LIN {X 0,Y 573.267,Z 626.574,A -85,B 0,C 180,E1 -2260.914,E2 -2260.914} C_VEL
LIN {X 0,Y 573.402,Z 606.241,A -85,B 0,C 180,E1 -2263.647,E2 -2263.647} C_VEL
LIN {X 0,Y 573.594,Z 585.071,A -85,B 0,C 180,E1 -2266.549,E2 -2266.549} C_VEL
LIN {X 0,Y 573.852,Z 562.818,A -85,B 0,C 180,E1 -2269.644,E2 -2269.644} C_VEL
LIN {X 0,Y 574.134,Z 540.047,A -85,B 0,C 180,E1 -2272.87,E2 -2272.87} C_VEL
LIN {X 0,Y 574.379,Z 520.07,A -85,B 0,C 180,E1 -2275.745,E2 -2275.745} C_VEL
LIN {X 0,Y 574.218,Z 508.518,A -85,B 0,C 180,E1 -2277.32,E2 -2277.32} C_VEL
LIN {X 0,Y 573.285,Z 503.963,A -85,B 0,C 180,E1 -2278.014,E2 -2278.014} C_VEL
LIN {X 0,Y 573.234,Z 503.898,A -85,B 0,C 180,E1 -2280.992,E2 -2280.992} C_VEL
LIN {X 0,Y 573.258,Z 503.887,A -85,B 0,C 180,E1 -2283.523,E2 -2283.523} C_VEL
LIN {X 0,Y 573.24,Z 503.887,A -85,B 0,C 180,E1 -2286.049,E2 -2286.049} C_VEL
LIN {X 0,Y 573.247,Z 503.892,A -85,B 0,C 180,E1 -2288.7,E2 -2288.7} C_VEL
LIN {X 0,Y 573.249,Z 503.887,A -85,B 0,C 180,E1 -2291.595,E2 -2291.595} C_VEL
LIN {X 0,Y 573.233,Z 503.889,A -85,B 0,C 180,E1 -2294.332,E2 -2294.332} C_VEL
LIN {X 0,Y 573.237,Z 503.89,A -85,B 0,C 180,E1 -2297.357,E2 -2297.357} C_VEL
LIN {X 0,Y 573.243,Z 503.888,A -85,B 0,C 180,E1 -2300.393,E2 -2300.393} C_VEL
LIN {X 0,Y 573.25,Z 503.892,A -85,B 0,C 180,E1 -2303.078,E2 -2303.078} C_VEL
LIN {X 0,Y 573.268,Z 503.884,A -85,B 0,C 180,E1 -2305.672,E2 -2305.672} C_VEL
LIN {X 0,Y 573.242,Z 503.886,A -85,B 0,C 180,E1 -2308.185,E2 -2308.185} C_VEL
LIN {X 0,Y 573.263,Z 503.889,A -85,B 0,C 180,E1 -2310.634,E2 -2310.634} C_VEL
LIN {X 0,Y 573.265,Z 503.884,A -85,B 0,C 180,E1 -2313.499,E2 -2313.499} C_VEL
LIN {X 0,Y 573.224,Z 503.889,A -85,B 0,C 180,E1 -2316.134,E2 -2316.134} C_VEL
LIN {X 0,Y 573.252,Z 503.89,A -85,B 0,C 180,E1 -2319.174,E2 -2319.174} C_VEL
LIN {X 0,Y 573.231,Z 503.89,A -85,B 0,C 180,E1 -2321.412,E2 -2321.412} C_VEL
LIN {X 0,Y 573.251,Z 503.886,A -85,B 0,C 180,E1 -2323.622,E2 -2323.622} C_VEL
LIN {X 0,Y 573.23,Z 503.893,A -85,B 0,C 180,E1 -2326.53,E2 -2326.53} C_VEL
LIN {X 0,Y 573.273,Z 503.891,A -85,B 0,C 180,E1 -2328.734,E2 -2328.734} C_VEL
LIN {X 0,Y 573.299,Z 503.881,A -85,B 0,C 180,E1 -2331.541,E2 -2331.541} C_VEL
LIN {X 0,Y 573.292,Z 503.883,A -85,B 0,C 180,E1 -2334.372,E2 -2334.372} C_VEL
LIN {X 0,Y 573.308,Z 503.883,A -85,B 0,C 180,E1 -2337.19,E2 -2337.19} C_VEL
LIN {X 0,Y 573.312,Z 503.879,A -85,B 0,C 180,E1 -2340,E2 -2340} C_VEL
LIN {X 0,Y 573.307,Z 503.888,A -85,B 0,C 180,E1 -2342.811,E2 -2342.811} C_VEL
LIN {X 0,Y 573.292,Z 503.883,A -85,B 0,C 180,E1 -2345.628,E2 -2345.628} C_VEL
LIN {X 0,Y 573.289,Z 503.968,A -85,B 0,C 180,E1 -2348.061,E2 -2348.061} C_VEL
LIN {X 0,Y 573.494,Z 504.97,A -85,B 0,C 180,E1 -2348.201,E2 -2348.201} C_VEL
LIN {X 0,Y 573.968,Z 507.089,A -85,B 0,C 180,E1 -2348.251,E2 -2348.251} C_VEL
LIN {X 0,Y 573.853,Z 535.33,A -85,B 0,C 180,E1 -2348.629,E2 -2348.629} C_VEL
LIN {X 0,Y 573.762,Z 548.888,A -85,B 0,C 180,E1 -2348.963,E2 -2348.963} C_VEL
LIN {X 0,Y 573.668,Z 561.556,A -85,B 0,C 180,E1 -2349.431,E2 -2349.431} C_VEL
LIN {X 0,Y 573.563,Z 572.433,A -85,B 0,C 180,E1 -2349.967,E2 -2349.967} C_VEL
LIN {X 0,Y 573.465,Z 582.587,A -85,B 0,C 180,E1 -2350.593,E2 -2350.593} C_VEL
LIN {X 0,Y 573.361,Z 592.106,A -85,B 0,C 180,E1 -2351.31,E2 -2351.31} C_VEL
LIN {X 0,Y 573.227,Z 601.905,A -85,B 0,C 180,E1 -2352.21,E2 -2352.21} C_VEL
LIN {X 0,Y 573.15,Z 611.329,A -85,B 0,C 180,E1 -2353.292,E2 -2353.292} C_VEL
LIN {X 0,Y 573.084,Z 618.697,A -85,B 0,C 180,E1 -2354.352,E2 -2354.352} C_VEL
LIN {X 0,Y 573.025,Z 624.017,A -85,B 0,C 180,E1 -2355.29,E2 -2355.29} C_VEL
LIN {X 0,Y 573.02,Z 626.025,A -85,B 0,C 180,E1 -2355.694,E2 -2355.694} C_VEL
LIN {X 0,Y 572.347,Z 628.414,A -85,B 0,C 180,E1 -2356.233,E2 -2356.233} C_VEL
LIN {X 0,Y 570.736,Z 630.55,A -85,B 0,C 180,E1 -2356.767,E2 -2356.767} C_VEL
LIN {X 0,Y 566.968,Z 633.967,A -85,B 0,C 180,E1 -2357.858,E2 -2357.858} C_VEL
LIN {X 0,Y 565.922,Z 635.258,A -85,B 0,C 180,E1 -2358.432,E2 -2358.432} C_VEL
LIN {X 0,Y 565.844,Z 635.651,A -85,B 0,C 180,E1 -2358.628,E2 -2358.628} C_VEL
LIN {X 0,Y 565.825,Z 637.129,A -85,B 0,C 180,E1 -2359.595,E2 -2359.595} C_VEL
LIN {X 0,Y 565.83,Z 637.763,A -85,B 0,C 180,E1 -2360.352,E2 -2360.352} C_VEL
LIN {X 0,Y 565.854,Z 637.935,A -85,B 0,C 180,E1 -2361.332,E2 -2361.332} C_VEL
LIN {X 0,Y 565.834,Z 636.939,A -85,B 0,C 180,E1 -2362.646,E2 -2362.646} C_VEL
LIN {X 0,Y 565.844,Z 635.773,A -85,B 0,C 180,E1 -2363.419,E2 -2363.419} C_VEL
LIN {X 0,Y 565.909,Z 633.01,A -85,B 0,C 180,E1 -2364.581,E2 -2364.581} C_VEL
LIN {X 0,Y 565.931,Z 628.982,A -85,B 0,C 180,E1 -2365.763,E2 -2365.763} C_VEL
LIN {X 0,Y 565.964,Z 623.586,A -85,B 0,C 180,E1 -2366.952,E2 -2366.952} C_VEL
LIN {X 0,Y 566.021,Z 617.865,A -85,B 0,C 180,E1 -2367.952,E2 -2367.952} C_VEL
LIN {X 0,Y 566.091,Z 610.807,A -85,B 0,C 180,E1 -2368.959,E2 -2368.959} C_VEL
LIN {X 0,Y 566.23,Z 601.095,A -85,B 0,C 180,E1 -2370.075,E2 -2370.075} C_VEL
LIN {X 0,Y 566.334,Z 591.882,A -85,B 0,C 180,E1 -2370.923,E2 -2370.923} C_VEL
LIN {X 0,Y 566.434,Z 582.793,A -85,B 0,C 180,E1 -2371.616,E2 -2371.616} C_VEL
LIN {X 0,Y 566.562,Z 572.874,A -85,B 0,C 180,E1 -2372.236,E2 -2372.236} C_VEL
LIN {X 0,Y 566.701,Z 562.695,A -85,B 0,C 180,E1 -2372.748,E2 -2372.748} C_VEL
LIN {X 0,Y 566.83,Z 552.002,A -85,B 0,C 180,E1 -2373.168,E2 -2373.168} C_VEL
LIN {X 0,Y 566.904,Z 541.21,A -85,B 0,C 180,E1 -2373.482,E2 -2373.482} C_VEL
LIN {X 0,Y 566.969,Z 529.772,A -85,B 0,C 180,E1 -2373.707,E2 -2373.707} C_VEL
LIN {X 0,Y 566.881,Z 507.314,A -85,B 0,C 180,E1 -2373.999,E2 -2373.999} C_VEL
LIN {X 0,Y 566.338,Z 505.338,A -85,B 0,C 180,E1 -2374.082,E2 -2374.082} C_VEL
LIN {X 0,Y 566.267,Z 504.787,A -85,B 0,C 180,E1 -2374.221,E2 -2374.221} C_VEL
LIN {X 0,Y 566.194,Z 504.774,A -85,B 0,C 180,E1 -2377.402,E2 -2377.402} C_VEL
LIN {X 0,Y 566.223,Z 504.761,A -85,B 0,C 180,E1 -2380.198,E2 -2380.198} C_VEL
LIN {X 0,Y 566.201,Z 504.769,A -85,B 0,C 180,E1 -2383.055,E2 -2383.055} C_VEL
LIN {X 0,Y 566.201,Z 504.764,A -85,B 0,C 180,E1 -2386.049,E2 -2386.049} C_VEL
LIN {X 0,Y 566.211,Z 504.764,A -85,B 0,C 180,E1 -2388.865,E2 -2388.865} C_VEL
LIN {X 0,Y 566.189,Z 504.771,A -85,B 0,C 180,E1 -2391.638,E2 -2391.638} C_VEL
LIN {X 0,Y 566.162,Z 504.768,A -85,B 0,C 180,E1 -2394.309,E2 -2394.309} C_VEL
LIN {X 0,Y 566.221,Z 504.762,A -85,B 0,C 180,E1 -2396.899,E2 -2396.899} C_VEL
LIN {X 0,Y 566.186,Z 504.774,A -85,B 0,C 180,E1 -2399.408,E2 -2399.408} C_VEL
LIN {X 0,Y 566.231,Z 504.764,A -85,B 0,C 180,E1 -2401.859,E2 -2401.859} C_VEL
LIN {X 0,Y 566.215,Z 504.762,A -85,B 0,C 180,E1 -2404.252,E2 -2404.252} C_VEL
LIN {X 0,Y 566.172,Z 504.767,A -85,B 0,C 180,E1 -2406.72,E2 -2406.72} C_VEL
LIN {X 0,Y 566.212,Z 504.77,A -85,B 0,C 180,E1 -2409.663,E2 -2409.663} C_VEL
LIN {X 0,Y 566.202,Z 504.763,A -85,B 0,C 180,E1 -2412.669,E2 -2412.669} C_VEL
LIN {X 0,Y 566.239,Z 504.769,A -85,B 0,C 180,E1 -2415.627,E2 -2415.627} C_VEL
LIN {X 0,Y 566.24,Z 504.758,A -85,B 0,C 180,E1 -2418.676,E2 -2418.676} C_VEL
LIN {X 0,Y 566.231,Z 504.765,A -85,B 0,C 180,E1 -2421.435,E2 -2421.435} C_VEL
LIN {X 0,Y 566.255,Z 504.758,A -85,B 0,C 180,E1 -2424.302,E2 -2424.302} C_VEL
LIN {X 0,Y 566.286,Z 504.76,A -85,B 0,C 180,E1 -2427.866,E2 -2427.866} C_VEL
LIN {X 0,Y 566.303,Z 504.75,A -85,B 0,C 180,E1 -2430.711,E2 -2430.711} C_VEL
LIN {X 0,Y 566.272,Z 504.754,A -85,B 0,C 180,E1 -2432.846,E2 -2432.846} C_VEL
LIN {X 0,Y 566.258,Z 504.765,A -85,B 0,C 180,E1 -2435.698,E2 -2435.698} C_VEL
LIN {X 0,Y 566.211,Z 504.762,A -85,B 0,C 180,E1 -2438.566,E2 -2438.566} C_VEL
LIN {X 0,Y 566.248,Z 504.761,A -85,B 0,C 180,E1 -2441.454,E2 -2441.454} C_VEL
LIN {X 0,Y 566.24,Z 504.759,A -85,B 0,C 180,E1 -2444.506,E2 -2444.506} C_VEL
LIN {X 0,Y 566.206,Z 504.764,A -85,B 0,C 180,E1 -2447.331,E2 -2447.331} C_VEL
LIN {X 0,Y 566.216,Z 504.764,A -85,B 0,C 180,E1 -2450.337,E2 -2450.337} C_VEL
LIN {X 0,Y 566.173,Z 504.768,A -85,B 0,C 180,E1 -2453.28,E2 -2453.28} C_VEL
LIN {X 0,Y 566.215,Z 504.768,A -85,B 0,C 180,E1 -2455.748,E2 -2455.748} C_VEL
LIN {X 0,Y 566.205,Z 504.769,A -85,B 0,C 180,E1 -2458.201,E2 -2458.201} C_VEL
LIN {X 0,Y 566.196,Z 504.763,A -85,B 0,C 180,E1 -2461.076,E2 -2461.076} C_VEL
LIN {X 0,Y 566.212,Z 504.767,A -85,B 0,C 180,E1 -2463.733,E2 -2463.733} C_VEL
LIN {X 0,Y 566.199,Z 504.765,A -85,B 0,C 180,E1 -2466.569,E2 -2466.569} C_VEL
LIN {X 0,Y 566.221,Z 504.761,A -85,B 0,C 180,E1 -2469.272,E2 -2469.272} C_VEL
LIN {X 0,Y 566.213,Z 504.772,A -85,B 0,C 180,E1 -2472.086,E2 -2472.086} C_VEL
LIN {X 0,Y 566.171,Z 504.767,A -85,B 0,C 180,E1 -2475.035,E2 -2475.035} C_VEL
LIN {X 0,Y 566.214,Z 504.772,A -85,B 0,C 180,E1 -2478.135,E2 -2478.135} C_VEL
LIN {X 0,Y 566.218,Z 504.763,A -85,B 0,C 180,E1 -2480.726,E2 -2480.726} C_VEL
LIN {X 0,Y 566.214,Z 504.765,A -85,B 0,C 180,E1 -2483.782,E2 -2483.782} C_VEL
LIN {X 0,Y 566.207,Z 504.772,A -85,B 0,C 180,E1 -2486.265,E2 -2486.265} C_VEL
LIN {X 0,Y 566.196,Z 504.764,A -85,B 0,C 180,E1 -2488.921,E2 -2488.921} C_VEL
LIN {X 0,Y 566.191,Z 504.764,A -85,B 0,C 180,E1 -2491.046,E2 -2491.046} C_VEL
LIN {X 0,Y 566.239,Z 504.758,A -85,B 0,C 180,E1 -2493.46,E2 -2493.46} C_VEL
LIN {X 0,Y 566.192,Z 504.767,A -85,B 0,C 180,E1 -2495.819,E2 -2495.819} C_VEL
LIN {X 0,Y 566.209,Z 504.764,A -85,B 0,C 180,E1 -2498.902,E2 -2498.902} C_VEL
LIN {X 0,Y 566.206,Z 504.762,A -85,B 0,C 180,E1 -2501.172,E2 -2501.172} C_VEL
LIN {X 0,Y 566.213,Z 504.761,A -85,B 0,C 180,E1 -2503.412,E2 -2503.412} C_VEL
LIN {X 0,Y 566.191,Z 504.775,A -85,B 0,C 180,E1 -2506.358,E2 -2506.358} C_VEL
LIN {X 0,Y 566.225,Z 504.765,A -85,B 0,C 180,E1 -2508.675,E2 -2508.675} C_VEL
LIN {X 0,Y 566.24,Z 504.758,A -85,B 0,C 180,E1 -2511.434,E2 -2511.434} C_VEL
LIN {X 0,Y 566.252,Z 504.765,A -85,B 0,C 180,E1 -2514.301,E2 -2514.301} C_VEL
LIN {X 0,Y 566.272,Z 504.756,A -85,B 0,C 180,E1 -2517.866,E2 -2517.866} C_VEL
LIN {X 0,Y 566.298,Z 504.757,A -85,B 0,C 180,E1 -2520.711,E2 -2520.711} C_VEL
LIN {X 0,Y 566.27,Z 504.759,A -85,B 0,C 180,E1 -2522.845,E2 -2522.845} C_VEL
LIN {X 0,Y 566.252,Z 504.757,A -85,B 0,C 180,E1 -2525.698,E2 -2525.698} C_VEL
LIN {X 0,Y 566.24,Z 504.769,A -85,B 0,C 180,E1 -2528.565,E2 -2528.565} C_VEL
LIN {X 0,Y 566.232,Z 504.759,A -85,B 0,C 180,E1 -2531.454,E2 -2531.454} C_VEL
LIN {X 0,Y 566.224,Z 504.769,A -85,B 0,C 180,E1 -2534.507,E2 -2534.507} C_VEL
LIN {X 0,Y 566.195,Z 504.765,A -85,B 0,C 180,E1 -2537.332,E2 -2537.332} C_VEL
LIN {X 0,Y 566.211,Z 504.767,A -85,B 0,C 180,E1 -2540.337,E2 -2540.337} C_VEL
LIN {X 0,Y 566.18,Z 504.766,A -85,B 0,C 180,E1 -2543.404,E2 -2543.404} C_VEL
LIN {X 0,Y 566.218,Z 504.761,A -85,B 0,C 180,E1 -2545.749,E2 -2545.749} C_VEL
LIN {X 0,Y 566.199,Z 504.766,A -85,B 0,C 180,E1 -2548.204,E2 -2548.204} C_VEL
LIN {X 0,Y 566.186,Z 504.773,A -85,B 0,C 180,E1 -2550.592,E2 -2550.592} C_VEL
LIN {X 0,Y 566.221,Z 504.765,A -85,B 0,C 180,E1 -2553.102,E2 -2553.102} C_VEL
LIN {X 0,Y 566.206,Z 504.762,A -85,B 0,C 180,E1 -2555.689,E2 -2555.689} C_VEL
LIN {X 0,Y 566.209,Z 504.768,A -85,B 0,C 180,E1 -2558.559,E2 -2558.559} C_VEL
LIN {X 0,Y 566.205,Z 504.767,A -85,B 0,C 180,E1 -2561.137,E2 -2561.137} C_VEL
LIN {X 0,Y 566.191,Z 504.764,A -85,B 0,C 180,E1 -2564.036,E2 -2564.036} C_VEL
LIN {X 0,Y 566.2,Z 504.77,A -85,B 0,C 180,E1 -2567.083,E2 -2567.083} C_VEL
LIN {X 0,Y 566.223,Z 504.76,A -85,B 0,C 180,E1 -2569.803,E2 -2569.803} C_VEL
LIN {X 0,Y 566.196,Z 504.768,A -85,B 0,C 180,E1 -2572.599,E2 -2572.599} C_VEL
LIN {X 0,Y 566.206,Z 504.77,A -85,B 0,C 180,E1 -2575.183,E2 -2575.183} C_VEL
LIN {X 0,Y 566.232,Z 504.762,A -85,B 0,C 180,E1 -2577.744,E2 -2577.744} C_VEL
LIN {X 0,Y 566.201,Z 504.768,A -85,B 0,C 180,E1 -2580.328,E2 -2580.328} C_VEL
LIN {X 0,Y 566.273,Z 504.993,A -85,B 0,C 180,E1 -2581.748,E2 -2581.748} C_VEL
LIN {X 0,Y 567.473,Z 511.299,A -85,B 0,C 180,E1 -2582.727,E2 -2582.727} C_VEL
LIN {X 0,Y 567.401,Z 525.917,A -85,B 0,C 180,E1 -2584.819,E2 -2584.819} C_VEL
LIN {X 0,Y 567.242,Z 541.371,A -85,B 0,C 180,E1 -2587.029,E2 -2587.029} C_VEL
LIN {X 0,Y 566.927,Z 561.23,A -85,B 0,C 180,E1 -2589.879,E2 -2589.879} C_VEL
LIN {X 0,Y 566.647,Z 582.435,A -85,B 0,C 180,E1 -2592.872,E2 -2592.872} C_VEL
LIN {X 0,Y 566.408,Z 604.916,A -85,B 0,C 180,E1 -2595.998,E2 -2595.998} C_VEL
LIN {X 0,Y 566.194,Z 626.308,A -85,B 0,C 180,E1 -2598.924,E2 -2598.924} C_VEL
LIN {X 0,Y 566.375,Z 628.043,A -85,B 0,C 180,E1 -2598.995,E2 -2598.995} C_VEL
LIN {X 0,Y 566.727,Z 637.345,A -85,B 0,C 180,E1 -2599.12,E2 -2599.12} C_VEL
LIN {X 0,Y 566.572,Z 704.153,A -85,B 0,C 180,E1 -2599.977,E2 -2599.977} C_VEL
LIN {X 0,Y 566.51,Z 713.427,A -85,B 0,C 180,E1 -2600.179,E2 -2600.179} C_VEL
LIN {X 0,Y 566.484,Z 721.901,A -85,B 0,C 180,E1 -2600.449,E2 -2600.449} C_VEL
LIN {X 0,Y 566.43,Z 730.403,A -85,B 0,C 180,E1 -2600.808,E2 -2600.808} C_VEL
LIN {X 0,Y 566.328,Z 738.734,A -85,B 0,C 180,E1 -2601.256,E2 -2601.256} C_VEL
LIN {X 0,Y 566.217,Z 746.774,A -85,B 0,C 180,E1 -2601.794,E2 -2601.794} C_VEL
LIN {X 0,Y 566.126,Z 755.436,A -85,B 0,C 180,E1 -2602.51,E2 -2602.51} C_VEL
LIN {X 0,Y 566.084,Z 763.926,A -85,B 0,C 180,E1 -2603.404,E2 -2603.404} C_VEL
LIN {X 0,Y 566.057,Z 769.434,A -85,B 0,C 180,E1 -2604.121,E2 -2604.121} C_VEL
LIN {X 0,Y 565.912,Z 774.988,A -85,B 0,C 180,E1 -2605.013,E2 -2605.013} C_VEL
LIN {X 0,Y 565.944,Z 780.148,A -85,B 0,C 180,E1 -2606.084,E2 -2606.084} C_VEL
LIN {X 0,Y 565.913,Z 782.788,A -85,B 0,C 180,E1 -2606.796,E2 -2606.796} C_VEL
LIN {X 0,Y 565.839,Z 785.681,A -85,B 0,C 180,E1 -2607.865,E2 -2607.865} C_VEL
LIN {X 0,Y 565.844,Z 786.935,A -85,B 0,C 180,E1 -2608.577,E2 -2608.577} C_VEL
LIN {X 0,Y 565.839,Z 787.71,A -85,B 0,C 180,E1 -2609.288,E2 -2609.288} C_VEL
LIN {X 0,Y 565.836,Z 788,A -85,B 0,C 180,E1 -2610,E2 -2610} C_VEL
LIN {X 0,Y 565.839,Z 787.711,A -85,B 0,C 180,E1 -2610.712,E2 -2610.712} C_VEL
LIN {X 0,Y 565.844,Z 786.936,A -85,B 0,C 180,E1 -2611.423,E2 -2611.423} C_VEL
LIN {X 0,Y 565.839,Z 785.683,A -85,B 0,C 180,E1 -2612.135,E2 -2612.135} C_VEL
LIN {X 0,Y 565.916,Z 782.789,A -85,B 0,C 180,E1 -2613.203,E2 -2613.203} C_VEL
LIN {X 0,Y 565.934,Z 780.148,A -85,B 0,C 180,E1 -2613.916,E2 -2613.916} C_VEL
LIN {X 0,Y 565.912,Z 774.989,A -85,B 0,C 180,E1 -2614.987,E2 -2614.987} C_VEL
LIN {X 0,Y 566.082,Z 768.191,A -85,B 0,C 180,E1 -2616.057,E2 -2616.057} C_VEL
LIN {X 0,Y 566.086,Z 761.251,A -85,B 0,C 180,E1 -2616.899,E2 -2616.899} C_VEL
LIN {X 0,Y 566.147,Z 753.409,A -85,B 0,C 180,E1 -2617.669,E2 -2617.669} C_VEL
LIN {X 0,Y 566.239,Z 745.548,A -85,B 0,C 180,E1 -2618.296,E2 -2618.296} C_VEL
LIN {X 0,Y 566.378,Z 735.735,A -85,B 0,C 180,E1 -2618.923,E2 -2618.923} C_VEL
LIN {X 0,Y 566.446,Z 724.309,A -85,B 0,C 180,E1 -2619.462,E2 -2619.462} C_VEL
LIN {X 0,Y 566.51,Z 714.256,A -85,B 0,C 180,E1 -2619.799,E2 -2619.799} C_VEL
LIN {X 0,Y 566.561,Z 705.459,A -85,B 0,C 180,E1 -2620.001,E2 -2620.001} C_VEL
LIN {X 0,Y 566.695,Z 653.576,A -85,B 0,C 180,E1 -2620.675,E2 -2620.675} C_VEL
LIN {X 0,Y 566.47,Z 628.888,A -85,B 0,C 180,E1 -2620.992,E2 -2620.992} C_VEL
LIN {X 0,Y 566.202,Z 626.566,A -85,B 0,C 180,E1 -2621.053,E2 -2621.053} C_VEL
LIN {X 0,Y 566.361,Z 607.565,A -85,B 0,C 180,E1 -2623.637,E2 -2623.637} C_VEL
LIN {X 0,Y 566.588,Z 586.383,A -85,B 0,C 180,E1 -2626.576,E2 -2626.576} C_VEL
LIN {X 0,Y 566.91,Z 564.011,A -85,B 0,C 180,E1 -2629.724,E2 -2629.724} C_VEL
LIN {X 0,Y 567.2,Z 542.695,A -85,B 0,C 180,E1 -2632.78,E2 -2632.78} C_VEL
LIN {X 0,Y 567.364,Z 529.068,A -85,B 0,C 180,E1 -2634.712,E2 -2634.712} C_VEL
LIN {X 0,Y 567.381,Z 512.067,A -85,B 0,C 180,E1 -2637.045,E2 -2637.045} C_VEL
LIN {X 0,Y 566.76,Z 507.496,A -85,B 0,C 180,E1 -2637.71,E2 -2637.71} C_VEL
LIN {X 0,Y 566.226,Z 504.819,A -85,B 0,C 180,E1 -2638.141,E2 -2638.141} C_VEL
LIN {X 0,Y 566.197,Z 504.773,A -85,B 0,C 180,E1 -2641.077,E2 -2641.077} C_VEL
LIN {X 0,Y 566.207,Z 504.764,A -85,B 0,C 180,E1 -2643.734,E2 -2643.734} C_VEL
LIN {X 0,Y 566.207,Z 504.767,A -85,B 0,C 180,E1 -2646.568,E2 -2646.568} C_VEL
LIN {X 0,Y 566.209,Z 504.763,A -85,B 0,C 180,E1 -2649.685,E2 -2649.685} C_VEL
LIN {X 0,Y 566.212,Z 504.762,A -85,B 0,C 180,E1 -2652.086,E2 -2652.086} C_VEL
LIN {X 0,Y 566.168,Z 504.777,A -85,B 0,C 180,E1 -2655.035,E2 -2655.035} C_VEL
LIN {X 0,Y 566.212,Z 504.761,A -85,B 0,C 180,E1 -2658.135,E2 -2658.135} C_VEL
LIN {X 0,Y 566.217,Z 504.768,A -85,B 0,C 180,E1 -2660.727,E2 -2660.727} C_VEL
LIN {X 0,Y 566.211,Z 504.762,A -85,B 0,C 180,E1 -2663.783,E2 -2663.783} C_VEL
LIN {X 0,Y 566.221,Z 504.762,A -85,B 0,C 180,E1 -2666.262,E2 -2666.262} C_VEL
LIN {X 0,Y 566.195,Z 504.774,A -85,B 0,C 180,E1 -2668.921,E2 -2668.921} C_VEL
LIN {X 0,Y 566.19,Z 504.773,A -85,B 0,C 180,E1 -2671.047,E2 -2671.047} C_VEL
LIN {X 0,Y 566.24,Z 504.76,A -85,B 0,C 180,E1 -2673.46,E2 -2673.46} C_VEL
LIN {X 0,Y 566.19,Z 504.765,A -85,B 0,C 180,E1 -2675.819,E2 -2675.819} C_VEL
LIN {X 0,Y 566.207,Z 504.772,A -85,B 0,C 180,E1 -2678.902,E2 -2678.902} C_VEL
LIN {X 0,Y 566.204,Z 504.768,A -85,B 0,C 180,E1 -2681.172,E2 -2681.172} C_VEL
LIN {X 0,Y 566.213,Z 504.764,A -85,B 0,C 180,E1 -2683.413,E2 -2683.413} C_VEL
LIN {X 0,Y 566.192,Z 504.767,A -85,B 0,C 180,E1 -2686.359,E2 -2686.359} C_VEL
LIN {X 0,Y 566.265,Z 504.762,A -85,B 0,C 180,E1 -2688.654,E2 -2688.654} C_VEL
LIN {X 0,Y 566.241,Z 504.761,A -85,B 0,C 180,E1 -2691.435,E2 -2691.435} C_VEL
LIN {X 0,Y 566.26,Z 504.759,A -85,B 0,C 180,E1 -2694.302,E2 -2694.302} C_VEL
LIN {X 0,Y 566.272,Z 504.755,A -85,B 0,C 180,E1 -2697.866,E2 -2697.866} C_VEL
LIN {X 0,Y 566.301,Z 504.76,A -85,B 0,C 180,E1 -2700.711,E2 -2700.711} C_VEL
LIN {X 0,Y 566.273,Z 504.765,A -85,B 0,C 180,E1 -2702.846,E2 -2702.846} C_VEL
LIN {X 0,Y 566.26,Z 504.759,A -85,B 0,C 180,E1 -2705.699,E2 -2705.699} C_VEL
LIN {X 0,Y 566.271,Z 504.99,A -85,B 0,C 180,E1 -2707.95,E2 -2707.95} C_VEL
LIN {X 0,Y 566.513,Z 506.087,A -85,B 0,C 180,E1 -2708.06,E2 -2708.06} C_VEL
LIN {X 0,Y 567.034,Z 508.715,A -85,B 0,C 180,E1 -2708.112,E2 -2708.112} C_VEL
LIN {X 0,Y 566.939,Z 535.503,A -85,B 0,C 180,E1 -2708.478,E2 -2708.478} C_VEL
LIN {X 0,Y 566.823,Z 549.345,A -85,B 0,C 180,E1 -2708.826,E2 -2708.826} C_VEL
LIN {X 0,Y 566.702,Z 561.368,A -85,B 0,C 180,E1 -2709.278,E2 -2709.278} C_VEL
LIN {X 0,Y 566.604,Z 572.262,A -85,B 0,C 180,E1 -2709.82,E2 -2709.82} C_VEL
LIN {X 0,Y 566.449,Z 582.465,A -85,B 0,C 180,E1 -2710.455,E2 -2710.455} C_VEL
LIN {X 0,Y 566.352,Z 591.303,A -85,B 0,C 180,E1 -2711.123,E2 -2711.123} C_VEL
LIN {X 0,Y 566.223,Z 599.052,A -85,B 0,C 180,E1 -2711.818,E2 -2711.818} C_VEL
LIN {X 0,Y 566.133,Z 605.977,A -85,B 0,C 180,E1 -2712.548,E2 -2712.548} C_VEL
LIN {X 0,Y 566.057,Z 613.271,A -85,B 0,C 180,E1 -2713.462,E2 -2713.462} C_VEL
LIN {X 0,Y 566.014,Z 619.63,A -85,B 0,C 180,E1 -2714.425,E2 -2714.425} C_VEL
LIN {X 0,Y 565.936,Z 625.335,A -85,B 0,C 180,E1 -2715.486,E2 -2715.486} C_VEL
LIN {X 0,Y 565.91,Z 630.045,A -85,B 0,C 180,E1 -2716.597,E2 -2716.597} C_VEL
LIN {X 0,Y 565.883,Z 633.608,A -85,B 0,C 180,E1 -2717.715,E2 -2717.715} C_VEL
LIN {X 0,Y 565.844,Z 635.651,A -85,B 0,C 180,E1 -2718.628,E2 -2718.628} C_VEL
LIN {X 0,Y 565.192,Z 636.695,A -85,B 0,C 180,E1 -2719.213,E2 -2719.213} C_VEL
LIN {X 0,Y 562.326,Z 637.702,A -85,B 0,C 180,E1 -2720.172,E2 -2720.172} C_VEL
LIN {X 0,Y 559.886,Z 637.985,A -85,B 0,C 180,E1 -2720.949,E2 -2720.949} C_VEL
LIN {X 0,Y 558.828,Z 637.836,A -85,B 0,C 180,E1 -2721.549,E2 -2721.549} C_VEL
LIN {X 0,Y 558.737,Z 637.727,A -85,B 0,C 180,E1 -2721.752,E2 -2721.752} C_VEL
LIN {X 0,Y 558.724,Z 636.569,A -85,B 0,C 180,E1 -2722.951,E2 -2722.951} C_VEL
LIN {X 0,Y 558.764,Z 635.221,A -85,B 0,C 180,E1 -2723.734,E2 -2723.734} C_VEL
LIN {X 0,Y 558.824,Z 633.314,A -85,B 0,C 180,E1 -2724.521,E2 -2724.521} C_VEL
LIN {X 0,Y 558.832,Z 629.408,A -85,B 0,C 180,E1 -2725.714,E2 -2725.714} C_VEL
LIN {X 0,Y 558.882,Z 624.859,A -85,B 0,C 180,E1 -2726.771,E2 -2726.771} C_VEL
LIN {X 0,Y 558.917,Z 619.769,A -85,B 0,C 180,E1 -2727.727,E2 -2727.727} C_VEL
LIN {X 0,Y 559.001,Z 613.117,A -85,B 0,C 180,E1 -2728.744,E2 -2728.744} C_VEL
LIN {X 0,Y 559.116,Z 605.655,A -85,B 0,C 180,E1 -2729.684,E2 -2729.684} C_VEL
LIN {X 0,Y 559.216,Z 597.973,A -85,B 0,C 180,E1 -2730.492,E2 -2730.492} C_VEL
LIN {X 0,Y 559.31,Z 590.476,A -85,B 0,C 180,E1 -2731.162,E2 -2731.162} C_VEL
LIN {X 0,Y 559.446,Z 581.356,A -85,B 0,C 180,E1 -2731.845,E2 -2731.845} C_VEL
LIN {X 0,Y 559.598,Z 573.039,A -85,B 0,C 180,E1 -2732.367,E2 -2732.367} C_VEL
LIN {X 0,Y 559.728,Z 563.251,A -85,B 0,C 180,E1 -2732.87,E2 -2732.87} C_VEL
LIN {X 0,Y 559.864,Z 553.819,A -85,B 0,C 180,E1 -2733.258,E2 -2733.258} C_VEL
LIN {X 0,Y 559.941,Z 542.6,A -85,B 0,C 180,E1 -2733.604,E2 -2733.604} C_VEL
LIN {X 0,Y 560.042,Z 531.139,A -85,B 0,C 180,E1 -2733.844,E2 -2733.844} C_VEL
LIN {X 0,Y 559.99,Z 508.607,A -85,B 0,C 180,E1 -2734.145,E2 -2734.145} C_VEL
LIN {X 0,Y 559.348,Z 506.397,A -85,B 0,C 180,E1 -2734.219,E2 -2734.219} C_VEL
LIN {X 0,Y 559.209,Z 505.671,A -85,B 0,C 180,E1 -2734.373,E2 -2734.373} C_VEL
LIN {X 0,Y 559.142,Z 505.652,A -85,B 0,C 180,E1 -2737.109,E2 -2737.109} C_VEL
LIN {X 0,Y 559.165,Z 505.642,A -85,B 0,C 180,E1 -2739.944,E2 -2739.944} C_VEL
LIN {X 0,Y 559.16,Z 505.642,A -85,B 0,C 180,E1 -2742.744,E2 -2742.744} C_VEL
LIN {X 0,Y 559.153,Z 505.645,A -85,B 0,C 180,E1 -2745.761,E2 -2745.761} C_VEL
LIN {X 0,Y 559.191,Z 505.636,A -85,B 0,C 180,E1 -2748.234,E2 -2748.234} C_VEL
LIN {X 0,Y 559.177,Z 505.644,A -85,B 0,C 180,E1 -2751.192,E2 -2751.192} C_VEL
LIN {X 0,Y 559.138,Z 505.647,A -85,B 0,C 180,E1 -2753.79,E2 -2753.79} C_VEL
LIN {X 0,Y 559.163,Z 505.64,A -85,B 0,C 180,E1 -2756.426,E2 -2756.426} C_VEL
LIN {X 0,Y 559.16,Z 505.643,A -85,B 0,C 180,E1 -2758.982,E2 -2758.982} C_VEL
LIN {X 0,Y 559.194,Z 505.636,A -85,B 0,C 180,E1 -2762.289,E2 -2762.289} C_VEL
LIN {X 0,Y 559.182,Z 505.638,A -85,B 0,C 180,E1 -2764.814,E2 -2764.814} C_VEL
LIN {X 0,Y 559.144,Z 505.647,A -85,B 0,C 180,E1 -2767.848,E2 -2767.848} C_VEL
LIN {X 0,Y 559.196,Z 505.635,A -85,B 0,C 180,E1 -2770.495,E2 -2770.495} C_VEL
LIN {X 0,Y 559.183,Z 505.641,A -85,B 0,C 180,E1 -2773.198,E2 -2773.198} C_VEL
LIN {X 0,Y 559.176,Z 505.64,A -85,B 0,C 180,E1 -2776.185,E2 -2776.185} C_VEL
LIN {X 0,Y 559.198,Z 505.638,A -85,B 0,C 180,E1 -2779.134,E2 -2779.134} C_VEL
LIN {X 0,Y 559.208,Z 505.638,A -85,B 0,C 180,E1 -2782.054,E2 -2782.054} C_VEL
LIN {X 0,Y 559.252,Z 505.629,A -85,B 0,C 180,E1 -2784.953,E2 -2784.953} C_VEL
LIN {X 0,Y 559.257,Z 505.636,A -85,B 0,C 180,E1 -2787.84,E2 -2787.84} C_VEL
LIN {X 0,Y 559.274,Z 505.626,A -85,B 0,C 180,E1 -2790.72,E2 -2790.72} C_VEL
LIN {X 0,Y 559.239,Z 505.63,A -85,B 0,C 180,E1 -2792.881,E2 -2792.881} C_VEL
LIN {X 0,Y 559.226,Z 505.642,A -85,B 0,C 180,E1 -2795.77,E2 -2795.77} C_VEL
LIN {X 0,Y 559.175,Z 505.638,A -85,B 0,C 180,E1 -2798.674,E2 -2798.674} C_VEL
LIN {X 0,Y 559.211,Z 505.64,A -85,B 0,C 180,E1 -2801.6,E2 -2801.6} C_VEL
LIN {X 0,Y 559.205,Z 505.635,A -85,B 0,C 180,E1 -2804.595,E2 -2804.595} C_VEL
LIN {X 0,Y 559.166,Z 505.644,A -85,B 0,C 180,E1 -2807.556,E2 -2807.556} C_VEL
LIN {X 0,Y 559.173,Z 505.648,A -85,B 0,C 180,E1 -2809.837,E2 -2809.837} C_VEL
LIN {X 0,Y 559.143,Z 505.648,A -85,B 0,C 180,E1 -2812.152,E2 -2812.152} C_VEL
LIN {X 0,Y 559.179,Z 505.639,A -85,B 0,C 180,E1 -2815.297,E2 -2815.297} C_VEL
LIN {X 0,Y 559.183,Z 505.643,A -85,B 0,C 180,E1 -2817.711,E2 -2817.711} C_VEL
LIN {X 0,Y 559.156,Z 505.647,A -85,B 0,C 180,E1 -2820.182,E2 -2820.182} C_VEL
LIN {X 0,Y 559.158,Z 505.641,A -85,B 0,C 180,E1 -2822.714,E2 -2822.714} C_VEL
LIN {X 0,Y 559.127,Z 505.645,A -85,B 0,C 180,E1 -2825.323,E2 -2825.323} C_VEL
LIN {X 0,Y 559.135,Z 505.653,A -85,B 0,C 180,E1 -2828.016,E2 -2828.016} C_VEL
LIN {X 0,Y 559.176,Z 505.639,A -85,B 0,C 180,E1 -2830.81,E2 -2830.81} C_VEL
LIN {X 0,Y 559.161,Z 505.644,A -85,B 0,C 180,E1 -2833.731,E2 -2833.731} C_VEL
LIN {X 0,Y 559.143,Z 505.643,A -85,B 0,C 180,E1 -2836.803,E2 -2836.803} C_VEL
LIN {X 0,Y 559.173,Z 505.638,A -85,B 0,C 180,E1 -2839.189,E2 -2839.189} C_VEL
LIN {X 0,Y 559.131,Z 505.651,A -85,B 0,C 180,E1 -2841.982,E2 -2841.982} C_VEL
LIN {X 0,Y 559.155,Z 505.642,A -85,B 0,C 180,E1 -2844.782,E2 -2844.782} C_VEL
LIN {X 0,Y 559.169,Z 505.639,A -85,B 0,C 180,E1 -2847.36,E2 -2847.36} C_VEL
LIN {X 0,Y 559.183,Z 505.646,A -85,B 0,C 180,E1 -2850.134,E2 -2850.134} C_VEL
LIN {X 0,Y 559.176,Z 505.638,A -85,B 0,C 180,E1 -2853.169,E2 -2853.169} C_VEL
LIN {X 0,Y 559.15,Z 505.642,A -85,B 0,C 180,E1 -2855.494,E2 -2855.494} C_VEL
LIN {X 0,Y 559.17,Z 505.644,A -85,B 0,C 180,E1 -2858.623,E2 -2858.623} C_VEL
LIN {X 0,Y 559.164,Z 505.641,A -85,B 0,C 180,E1 -2860.926,E2 -2860.926} C_VEL
LIN {X 0,Y 559.163,Z 505.643,A -85,B 0,C 180,E1 -2863.947,E2 -2863.947} C_VEL
LIN {X 0,Y 559.165,Z 505.646,A -85,B 0,C 180,E1 -2866.184,E2 -2866.184} C_VEL
LIN {X 0,Y 559.187,Z 505.637,A -85,B 0,C 180,E1 -2869.133,E2 -2869.133} C_VEL
LIN {X 0,Y 559.202,Z 505.639,A -85,B 0,C 180,E1 -2872.053,E2 -2872.053} C_VEL
LIN {X 0,Y 559.251,Z 505.631,A -85,B 0,C 180,E1 -2874.953,E2 -2874.953} C_VEL
LIN {X 0,Y 559.244,Z 505.631,A -85,B 0,C 180,E1 -2877.839,E2 -2877.839} C_VEL
LIN {X 0,Y 559.268,Z 505.633,A -85,B 0,C 180,E1 -2880.72,E2 -2880.72} C_VEL
LIN {X 0,Y 559.236,Z 505.635,A -85,B 0,C 180,E1 -2882.881,E2 -2882.881} C_VEL
LIN {X 0,Y 559.221,Z 505.633,A -85,B 0,C 180,E1 -2885.77,E2 -2885.77} C_VEL
LIN {X 0,Y 559.194,Z 505.644,A -85,B 0,C 180,E1 -2888.674,E2 -2888.674} C_VEL
LIN {X 0,Y 559.195,Z 505.636,A -85,B 0,C 180,E1 -2891.6,E2 -2891.6} C_VEL
LIN {X 0,Y 559.189,Z 505.647,A -85,B 0,C 180,E1 -2894.596,E2 -2894.596} C_VEL
LIN {X 0,Y 559.155,Z 505.641,A -85,B 0,C 180,E1 -2897.557,E2 -2897.557} C_VEL
LIN {X 0,Y 559.166,Z 505.64,A -85,B 0,C 180,E1 -2899.837,E2 -2899.837} C_VEL
LIN {X 0,Y 559.134,Z 505.646,A -85,B 0,C 180,E1 -2902.153,E2 -2902.153} C_VEL
LIN {X 0,Y 559.171,Z 505.641,A -85,B 0,C 180,E1 -2905.188,E2 -2905.188} C_VEL
LIN {X 0,Y 559.186,Z 505.637,A -85,B 0,C 180,E1 -2907.712,E2 -2907.712} C_VEL
LIN {X 0,Y 559.161,Z 505.642,A -85,B 0,C 180,E1 -2910.182,E2 -2910.182} C_VEL
LIN {X 0,Y 559.168,Z 505.649,A -85,B 0,C 180,E1 -2912.714,E2 -2912.714} C_VEL
LIN {X 0,Y 559.152,Z 505.643,A -85,B 0,C 180,E1 -2915.322,E2 -2915.322} C_VEL
LIN {X 0,Y 559.128,Z 505.644,A -85,B 0,C 180,E1 -2918.018,E2 -2918.018} C_VEL
LIN {X 0,Y 559.17,Z 505.649,A -85,B 0,C 180,E1 -2920.811,E2 -2920.811} C_VEL
LIN {X 0,Y 559.135,Z 505.643,A -85,B 0,C 180,E1 -2923.734,E2 -2923.734} C_VEL
LIN {X 0,Y 559.163,Z 505.649,A -85,B 0,C 180,E1 -2926.802,E2 -2926.802} C_VEL
LIN {X 0,Y 559.172,Z 505.644,A -85,B 0,C 180,E1 -2929.19,E2 -2929.19} C_VEL
LIN {X 0,Y 559.132,Z 505.643,A -85,B 0,C 180,E1 -2931.983,E2 -2931.983} C_VEL
LIN {X 0,Y 559.143,Z 505.651,A -85,B 0,C 180,E1 -2934.785,E2 -2934.785} C_VEL
LIN {X 0,Y 559.172,Z 505.645,A -85,B 0,C 180,E1 -2937.362,E2 -2937.362} C_VEL
LIN {X 0,Y 559.147,Z 505.646,A -85,B 0,C 180,E1 -2940.143,E2 -2940.143} C_VEL
LIN {X 0,Y 559.197,Z 505.759,A -85,B 0,C 180,E1 -2941.527,E2 -2941.527} C_VEL
LIN {X 0,Y 560.577,Z 513.132,A -85,B 0,C 180,E1 -2942.706,E2 -2942.706} C_VEL
LIN {X 0,Y 560.436,Z 530.107,A -85,B 0,C 180,E1 -2945.16,E2 -2945.16} C_VEL
LIN {X 0,Y 560.273,Z 547.955,A -85,B 0,C 180,E1 -2947.701,E2 -2947.701} C_VEL
LIN {X 0,Y 559.879,Z 568.241,A -85,B 0,C 180,E1 -2950.628,E2 -2950.628} C_VEL
LIN {X 0,Y 559.611,Z 587.706,A -85,B 0,C 180,E1 -2953.399,E2 -2953.399} C_VEL
LIN {X 0,Y 559.333,Z 608.888,A -85,B 0,C 180,E1 -2956.374,E2 -2956.374} C_VEL
LIN {X 0,Y 559.172,Z 626.556,A -85,B 0,C 180,E1 -2958.802,E2 -2958.802} C_VEL
LIN {X 0,Y 559.721,Z 631.705,A -85,B 0,C 180,E1 -2958.91,E2 -2958.91} C_VEL
LIN {X 0,Y 559.598,Z 704.153,A -85,B 0,C 180,E1 -2959.851,E2 -2959.851} C_VEL
LIN {X 0,Y 559.524,Z 713.427,A -85,B 0,C 180,E1 -2960.055,E2 -2960.055} C_VEL
LIN {X 0,Y 559.493,Z 721.9,A -85,B 0,C 180,E1 -2960.328,E2 -2960.328} C_VEL
LIN {X 0,Y 559.434,Z 730.401,A -85,B 0,C 180,E1 -2960.692,E2 -2960.692} C_VEL
LIN {X 0,Y 559.303,Z 738.732,A -85,B 0,C 180,E1 -2961.145,E2 -2961.145} C_VEL
LIN {X 0,Y 559.183,Z 746.776,A -85,B 0,C 180,E1 -2961.69,E2 -2961.69} C_VEL
LIN {X 0,Y 559.096,Z 755.437,A -85,B 0,C 180,E1 -2962.416,E2 -2962.416} C_VEL
LIN {X 0,Y 559.03,Z 763.756,A -85,B 0,C 180,E1 -2963.299,E2 -2963.299} C_VEL
LIN {X 0,Y 559.004,Z 769.435,A -85,B 0,C 180,E1 -2964.047,E2 -2964.047} C_VEL
LIN {X 0,Y 558.826,Z 774.988,A -85,B 0,C 180,E1 -2964.95,E2 -2964.95} C_VEL
LIN {X 0,Y 558.859,Z 780.149,A -85,B 0,C 180,E1 -2966.034,E2 -2966.034} C_VEL
LIN {X 0,Y 558.805,Z 783.935,A -85,B 0,C 180,E1 -2967.116,E2 -2967.116} C_VEL
LIN {X 0,Y 558.745,Z 785.682,A -85,B 0,C 180,E1 -2967.837,E2 -2967.837} C_VEL
LIN {X 0,Y 558.744,Z 786.934,A -85,B 0,C 180,E1 -2968.558,E2 -2968.558} C_VEL
LIN {X 0,Y 558.739,Z 787.709,A -85,B 0,C 180,E1 -2969.279,E2 -2969.279} C_VEL
LIN {X 0,Y 558.737,Z 788,A -85,B 0,C 180,E1 -2970,E2 -2970} C_VEL
LIN {X 0,Y 558.739,Z 787.71,A -85,B 0,C 180,E1 -2970.721,E2 -2970.721} C_VEL
LIN {X 0,Y 558.744,Z 786.935,A -85,B 0,C 180,E1 -2971.441,E2 -2971.441} C_VEL
LIN {X 0,Y 558.745,Z 785.683,A -85,B 0,C 180,E1 -2972.162,E2 -2972.162} C_VEL
LIN {X 0,Y 558.841,Z 782.789,A -85,B 0,C 180,E1 -2973.244,E2 -2973.244} C_VEL
LIN {X 0,Y 558.851,Z 780.148,A -85,B 0,C 180,E1 -2973.966,E2 -2973.966} C_VEL
LIN {X 0,Y 558.826,Z 774.99,A -85,B 0,C 180,E1 -2975.05,E2 -2975.05} C_VEL
LIN {X 0,Y 559.007,Z 768.19,A -85,B 0,C 180,E1 -2976.134,E2 -2976.134} C_VEL
LIN {X 0,Y 559.045,Z 760.747,A -85,B 0,C 180,E1 -2977.04,E2 -2977.04} C_VEL
LIN {X 0,Y 559.121,Z 753.407,A -85,B 0,C 180,E1 -2977.766,E2 -2977.766} C_VEL
LIN {X 0,Y 559.222,Z 745.546,A -85,B 0,C 180,E1 -2978.401,E2 -2978.401} C_VEL
LIN {X 0,Y 559.36,Z 735.734,A -85,B 0,C 180,E1 -2979.036,E2 -2979.036} C_VEL
LIN {X 0,Y 559.436,Z 724.311,A -85,B 0,C 180,E1 -2979.581,E2 -2979.581} C_VEL
LIN {X 0,Y 559.518,Z 714.256,A -85,B 0,C 180,E1 -2979.922,E2 -2979.922} C_VEL
LIN {X 0,Y 559.569,Z 705.458,A -85,B 0,C 180,E1 -2980.127,E2 -2980.127} C_VEL
LIN {X 0,Y 559.66,Z 667.885,A -85,B 0,C 180,E1 -2980.628,E2 -2980.628} C_VEL
LIN {X 0,Y 559.544,Z 629.63,A -85,B 0,C 180,E1 -2981.12,E2 -2981.12} C_VEL
LIN {X 0,Y 559.176,Z 626.543,A -85,B 0,C 180,E1 -2981.196,E2 -2981.196} C_VEL
LIN {X 0,Y 559.383,Z 606.241,A -85,B 0,C 180,E1 -2983.996,E2 -2983.996} C_VEL
LIN {X 0,Y 559.688,Z 583.114,A -85,B 0,C 180,E1 -2987.251,E2 -2987.251} C_VEL
LIN {X 0,Y 559.988,Z 562.553,A -85,B 0,C 180,E1 -2990.189,E2 -2990.189} C_VEL
LIN {X 0,Y 560.286,Z 545.171,A -85,B 0,C 180,E1 -2992.688,E2 -2992.688} C_VEL
LIN {X 0,Y 560.375,Z 526.529,A -85,B 0,C 180,E1 -2995.24,E2 -2995.24} C_VEL
LIN {X 0,Y 560.381,Z 511.744,A -85,B 0,C 180,E1 -2997.318,E2 -2997.318} C_VEL
LIN {X 0,Y 559.214,Z 505.846,A -85,B 0,C 180,E1 -2998.212,E2 -2998.212} C_VEL
LIN {X 0,Y 559.151,Z 505.648,A -85,B 0,C 180,E1 -3001.274,E2 -3001.274} C_VEL
LIN {X 0,Y 559.162,Z 505.642,A -85,B 0,C 180,E1 -3003.949,E2 -3003.949} C_VEL
LIN {X 0,Y 559.142,Z 505.651,A -85,B 0,C 180,E1 -3007.107,E2 -3007.107} C_VEL
LIN {X 0,Y 559.165,Z 505.64,A -85,B 0,C 180,E1 -3009.942,E2 -3009.942} C_VEL
LIN {X 0,Y 559.163,Z 505.647,A -85,B 0,C 180,E1 -3012.742,E2 -3012.742} C_VEL
LIN {X 0,Y 559.149,Z 505.642,A -85,B 0,C 180,E1 -3015.76,E2 -3015.76} C_VEL
LIN {X 0,Y 559.185,Z 505.637,A -85,B 0,C 180,E1 -3018.232,E2 -3018.232} C_VEL
LIN {X 0,Y 559.172,Z 505.645,A -85,B 0,C 180,E1 -3021.19,E2 -3021.19} C_VEL
LIN {X 0,Y 559.166,Z 505.639,A -85,B 0,C 180,E1 -3023.791,E2 -3023.791} C_VEL
LIN {X 0,Y 559.17,Z 505.642,A -85,B 0,C 180,E1 -3026.426,E2 -3026.426} C_VEL
LIN {X 0,Y 559.159,Z 505.65,A -85,B 0,C 180,E1 -3028.981,E2 -3028.981} C_VEL
LIN {X 0,Y 559.162,Z 505.641,A -85,B 0,C 180,E1 -3031.618,E2 -3031.618} C_VEL
LIN {X 0,Y 559.193,Z 505.635,A -85,B 0,C 180,E1 -3033.904,E2 -3033.904} C_VEL
LIN {X 0,Y 559.148,Z 505.647,A -85,B 0,C 180,E1 -3036.567,E2 -3036.567} C_VEL
LIN {X 0,Y 559.177,Z 505.641,A -85,B 0,C 180,E1 -3039.396,E2 -3039.396} C_VEL
LIN {X 0,Y 559.146,Z 505.642,A -85,B 0,C 180,E1 -3041.686,E2 -3041.686} C_VEL
LIN {X 0,Y 559.163,Z 505.64,A -85,B 0,C 180,E1 -3043.948,E2 -3043.948} C_VEL
LIN {X 0,Y 559.165,Z 505.641,A -85,B 0,C 180,E1 -3046.184,E2 -3046.184} C_VEL
LIN {X 0,Y 559.202,Z 505.642,A -85,B 0,C 180,E1 -3049.134,E2 -3049.134} C_VEL
LIN {X 0,Y 559.205,Z 505.636,A -85,B 0,C 180,E1 -3052.054,E2 -3052.054} C_VEL
LIN {X 0,Y 559.254,Z 505.638,A -85,B 0,C 180,E1 -3054.954,E2 -3054.954} C_VEL
LIN {X 0,Y 559.244,Z 505.631,A -85,B 0,C 180,E1 -3057.84,E2 -3057.84} C_VEL
LIN {X 0,Y 559.27,Z 505.636,A -85,B 0,C 180,E1 -3060.72,E2 -3060.72} C_VEL
LIN {X 0,Y 559.239,Z 505.64,A -85,B 0,C 180,E1 -3062.882,E2 -3062.882} C_VEL
LIN {X 0,Y 559.23,Z 505.635,A -85,B 0,C 180,E1 -3065.77,E2 -3065.77} C_VEL
LIN {X 0,Y 559.21,Z 505.761,A -85,B 0,C 180,E1 -3067.765,E2 -3067.765} C_VEL
LIN {X 0,Y 559.443,Z 506.789,A -85,B 0,C 180,E1 -3067.898,E2 -3067.898} C_VEL
LIN {X 0,Y 560.12,Z 509.224,A -85,B 0,C 180,E1 -3067.956,E2 -3067.956} C_VEL
LIN {X 0,Y 560.022,Z 535.514,A -85,B 0,C 180,E1 -3068.321,E2 -3068.321} C_VEL
LIN {X 0,Y 559.903,Z 549.033,A -85,B 0,C 180,E1 -3068.663,E2 -3068.663} C_VEL
LIN {X 0,Y 559.751,Z 561.171,A -85,B 0,C 180,E1 -3069.121,E2 -3069.121} C_VEL
LIN {X 0,Y 559.637,Z 572.099,A -85,B 0,C 180,E1 -3069.67,E2 -3069.67} C_VEL
LIN {X 0,Y 559.482,Z 581.031,A -85,B 0,C 180,E1 -3070.221,E2 -3070.221} C_VEL
LIN {X 0,Y 559.351,Z 589.702,A -85,B 0,C 180,E1 -3070.864,E2 -3070.864} C_VEL
LIN {X 0,Y 559.22,Z 598.027,A -85,B 0,C 180,E1 -3071.6,E2 -3071.6} C_VEL
LIN {X 0,Y 559.118,Z 605.107,A -85,B 0,C 180,E1 -3072.339,E2 -3072.339} C_VEL
LIN {X 0,Y 559.008,Z 612.538,A -85,B 0,C 180,E1 -3073.265,E2 -3073.265} C_VEL
LIN {X 0,Y 558.959,Z 618.531,A -85,B 0,C 180,E1 -3074.158,E2 -3074.158} C_VEL
LIN {X 0,Y 558.914,Z 622.992,A -85,B 0,C 180,E1 -3074.938,E2 -3074.938} C_VEL
LIN {X 0,Y 558.829,Z 628.174,A -85,B 0,C 180,E1 -3076.062,E2 -3076.062} C_VEL
LIN {X 0,Y 558.801,Z 631.888,A -85,B 0,C 180,E1 -3077.094,E2 -3077.094} C_VEL
LIN {X 0,Y 558.744,Z 635.101,A -85,B 0,C 180,E1 -3078.328,E2 -3078.328} C_VEL
LIN {X 0,Y 558.759,Z 636.879,A -85,B 0,C 180,E1 -3079.384,E2 -3079.384} C_VEL
LIN {X 0,Y 558.738,Z 637.871,A -85,B 0,C 180,E1 -3080.622,E2 -3080.622} C_VEL
LIN {X 0,Y 558.737,Z 637.727,A -85,B 0,C 180,E1 -3081.752,E2 -3081.752} C_VEL
LIN {X 0,Y 558.065,Z 637.333,A -85,B 0,C 180,E1 -3082.353,E2 -3082.353} C_VEL
LIN {X 0,Y 555.242,Z 636.044,A -85,B 0,C 180,E1 -3083.322,E2 -3083.322} C_VEL
LIN {X 0,Y 552.86,Z 634.489,A -85,B 0,C 180,E1 -3084.092,E2 -3084.092} C_VEL
LIN {X 0,Y 551.83,Z 632.982,A -85,B 0,C 180,E1 -3084.678,E2 -3084.678} C_VEL
LIN {X 0,Y 551.741,Z 632.384,A -85,B 0,C 180,E1 -3084.875,E2 -3084.875} C_VEL
LIN {X 0,Y 551.754,Z 628.239,A -85,B 0,C 180,E1 -3086.069,E2 -3086.069} C_VEL
LIN {X 0,Y 551.805,Z 624.409,A -85,B 0,C 180,E1 -3086.935,E2 -3086.935} C_VEL
LIN {X 0,Y 551.868,Z 619.198,A -85,B 0,C 180,E1 -3087.905,E2 -3087.905} C_VEL
LIN {X 0,Y 551.936,Z 614.164,A -85,B 0,C 180,E1 -3088.698,E2 -3088.698} C_VEL
LIN {X 0,Y 552.056,Z 607.684,A -85,B 0,C 180,E1 -3089.559,E2 -3089.559} C_VEL
LIN {X 0,Y 552.18,Z 599.644,A -85,B 0,C 180,E1 -3090.449,E2 -3090.449} C_VEL
LIN {X 0,Y 552.287,Z 591.139,A -85,B 0,C 180,E1 -3091.236,E2 -3091.236} C_VEL
LIN {X 0,Y 552.446,Z 581.922,A -85,B 0,C 180,E1 -3091.944,E2 -3091.944} C_VEL
LIN {X 0,Y 552.632,Z 573.338,A -85,B 0,C 180,E1 -3092.493,E2 -3092.493} C_VEL
LIN {X 0,Y 552.773,Z 563.566,A -85,B 0,C 180,E1 -3093.006,E2 -3093.006} C_VEL
LIN {X 0,Y 552.911,Z 554.067,A -85,B 0,C 180,E1 -3093.405,E2 -3093.405} C_VEL
LIN {X 0,Y 553.008,Z 543.023,A -85,B 0,C 180,E1 -3093.753,E2 -3093.753} C_VEL
LIN {X 0,Y 553.129,Z 532.015,A -85,B 0,C 180,E1 -3093.991,E2 -3093.991} C_VEL
LIN {X 0,Y 553.162,Z 510.197,A -85,B 0,C 180,E1 -3094.289,E2 -3094.289} C_VEL
LIN {X 0,Y 552.299,Z 507.282,A -85,B 0,C 180,E1 -3094.379,E2 -3094.379} C_VEL
LIN {X 0,Y 552.188,Z 506.553,A -85,B 0,C 180,E1 -3094.523,E2 -3094.523} C_VEL
LIN {X 0,Y 552.089,Z 506.528,A -85,B 0,C 180,E1 -3097.665,E2 -3097.665} C_VEL
LIN {X 0,Y 552.118,Z 506.519,A -85,B 0,C 180,E1 -3100.481,E2 -3100.481} C_VEL
LIN {X 0,Y 552.111,Z 506.527,A -85,B 0,C 180,E1 -3103.485,E2 -3103.485} C_VEL
LIN {X 0,Y 552.12,Z 506.517,A -85,B 0,C 180,E1 -3106.579,E2 -3106.579} C_VEL
LIN {X 0,Y 552.141,Z 506.523,A -85,B 0,C 180,E1 -3109.523,E2 -3109.523} C_VEL
LIN {X 0,Y 552.093,Z 506.52,A -85,B 0,C 180,E1 -3112.337,E2 -3112.337} C_VEL
LIN {X 0,Y 552.084,Z 506.525,A -85,B 0,C 180,E1 -3115.052,E2 -3115.052} C_VEL
LIN {X 0,Y 552.127,Z 506.523,A -85,B 0,C 180,E1 -3117.683,E2 -3117.683} C_VEL
LIN {X 0,Y 552.113,Z 506.518,A -85,B 0,C 180,E1 -3120.236,E2 -3120.236} C_VEL
LIN {X 0,Y 552.143,Z 506.517,A -85,B 0,C 180,E1 -3123,E2 -3123} C_VEL
LIN {X 0,Y 552.116,Z 506.522,A -85,B 0,C 180,E1 -3125.162,E2 -3125.162} C_VEL
LIN {X 0,Y 552.129,Z 506.516,A -85,B 0,C 180,E1 -3128.338,E2 -3128.338} C_VEL
LIN {X 0,Y 552.154,Z 506.513,A -85,B 0,C 180,E1 -3130.675,E2 -3130.675} C_VEL
LIN {X 0,Y 552.118,Z 506.525,A -85,B 0,C 180,E1 -3133.738,E2 -3133.738} C_VEL
LIN {X 0,Y 552.14,Z 506.519,A -85,B 0,C 180,E1 -3136.005,E2 -3136.005} C_VEL
LIN {X 0,Y 552.166,Z 506.512,A -85,B 0,C 180,E1 -3138.994,E2 -3138.994} C_VEL
LIN {X 0,Y 552.162,Z 506.517,A -85,B 0,C 180,E1 -3141.952,E2 -3141.952} C_VEL
LIN {X 0,Y 552.227,Z 506.504,A -85,B 0,C 180,E1 -3144.889,E2 -3144.889} C_VEL
LIN {X 0,Y 552.228,Z 506.512,A -85,B 0,C 180,E1 -3147.812,E2 -3147.812} C_VEL
LIN {X 0,Y 552.244,Z 506.501,A -85,B 0,C 180,E1 -3150.729,E2 -3150.729} C_VEL
LIN {X 0,Y 552.206,Z 506.506,A -85,B 0,C 180,E1 -3152.918,E2 -3152.918} C_VEL
LIN {X 0,Y 552.195,Z 506.517,A -85,B 0,C 180,E1 -3155.844,E2 -3155.844} C_VEL
LIN {X 0,Y 552.15,Z 506.513,A -85,B 0,C 180,E1 -3158.786,E2 -3158.786} C_VEL
LIN {X 0,Y 552.168,Z 506.52,A -85,B 0,C 180,E1 -3161.75,E2 -3161.75} C_VEL
LIN {X 0,Y 552.141,Z 506.514,A -85,B 0,C 180,E1 -3164.748,E2 -3164.748} C_VEL
LIN {X 0,Y 552.116,Z 506.526,A -85,B 0,C 180,E1 -3167.788,E2 -3167.788} C_VEL
LIN {X 0,Y 552.133,Z 506.522,A -85,B 0,C 180,E1 -3170.101,E2 -3170.101} C_VEL
LIN {X 0,Y 552.095,Z 506.522,A -85,B 0,C 180,E1 -3172.45,E2 -3172.45} C_VEL
LIN {X 0,Y 552.158,Z 506.514,A -85,B 0,C 180,E1 -3175.35,E2 -3175.35} C_VEL
LIN {X 0,Y 552.122,Z 506.525,A -85,B 0,C 180,E1 -3178.097,E2 -3178.097} C_VEL
LIN {X 0,Y 552.106,Z 506.52,A -85,B 0,C 180,E1 -3180.608,E2 -3180.608} C_VEL
LIN {X 0,Y 552.116,Z 506.518,A -85,B 0,C 180,E1 -3183.185,E2 -3183.185} C_VEL
LIN {X 0,Y 552.085,Z 506.528,A -85,B 0,C 180,E1 -3185.843,E2 -3185.843} C_VEL
LIN {X 0,Y 552.125,Z 506.516,A -85,B 0,C 180,E1 -3189.061,E2 -3189.061} C_VEL
LIN {X 0,Y 552.139,Z 506.516,A -85,B 0,C 180,E1 -3191.443,E2 -3191.443} C_VEL
LIN {X 0,Y 552.094,Z 506.524,A -85,B 0,C 180,E1 -3194.531,E2 -3194.531} C_VEL
LIN {X 0,Y 552.128,Z 506.518,A -85,B 0,C 180,E1 -3197.584,E2 -3197.584} C_VEL
LIN {X 0,Y 552.131,Z 506.521,A -85,B 0,C 180,E1 -3200.472,E2 -3200.472} C_VEL
LIN {X 0,Y 552.11,Z 506.518,A -85,B 0,C 180,E1 -3203.315,E2 -3203.315} C_VEL
LIN {X 0,Y 552.127,Z 506.522,A -85,B 0,C 180,E1 -3205.939,E2 -3205.939} C_VEL
LIN {X 0,Y 552.113,Z 506.523,A -85,B 0,C 180,E1 -3208.54,E2 -3208.54} C_VEL
LIN {X 0,Y 552.12,Z 506.517,A -85,B 0,C 180,E1 -3211.437,E2 -3211.437} C_VEL
LIN {X 0,Y 552.131,Z 506.524,A -85,B 0,C 180,E1 -3214.355,E2 -3214.355} C_VEL
LIN {X 0,Y 552.103,Z 506.522,A -85,B 0,C 180,E1 -3216.758,E2 -3216.758} C_VEL
LIN {X 0,Y 552.119,Z 506.517,A -85,B 0,C 180,E1 -3219.119,E2 -3219.119} C_VEL
LIN {X 0,Y 552.124,Z 506.517,A -85,B 0,C 180,E1 -3221.444,E2 -3221.444} C_VEL
LIN {X 0,Y 552.112,Z 506.519,A -85,B 0,C 180,E1 -3223.737,E2 -3223.737} C_VEL
LIN {X 0,Y 552.128,Z 506.52,A -85,B 0,C 180,E1 -3226.004,E2 -3226.004} C_VEL
LIN {X 0,Y 552.154,Z 506.514,A -85,B 0,C 180,E1 -3228.993,E2 -3228.993} C_VEL
LIN {X 0,Y 552.156,Z 506.516,A -85,B 0,C 180,E1 -3231.951,E2 -3231.951} C_VEL
LIN {X 0,Y 552.225,Z 506.507,A -85,B 0,C 180,E1 -3234.889,E2 -3234.889} C_VEL
LIN {X 0,Y 552.215,Z 506.506,A -85,B 0,C 180,E1 -3237.812,E2 -3237.812} C_VEL
LIN {X 0,Y 552.237,Z 506.508,A -85,B 0,C 180,E1 -3240.729,E2 -3240.729} C_VEL
LIN {X 0,Y 552.202,Z 506.51,A -85,B 0,C 180,E1 -3242.918,E2 -3242.918} C_VEL
LIN {X 0,Y 552.191,Z 506.509,A -85,B 0,C 180,E1 -3245.844,E2 -3245.844} C_VEL
LIN {X 0,Y 552.162,Z 506.518,A -85,B 0,C 180,E1 -3248.785,E2 -3248.785} C_VEL
LIN {X 0,Y 552.153,Z 506.513,A -85,B 0,C 180,E1 -3251.75,E2 -3251.75} C_VEL
LIN {X 0,Y 552.127,Z 506.524,A -85,B 0,C 180,E1 -3254.748,E2 -3254.748} C_VEL
LIN {X 0,Y 552.106,Z 506.519,A -85,B 0,C 180,E1 -3257.788,E2 -3257.788} C_VEL
LIN {X 0,Y 552.125,Z 506.518,A -85,B 0,C 180,E1 -3260.101,E2 -3260.101} C_VEL
LIN {X 0,Y 552.088,Z 506.527,A -85,B 0,C 180,E1 -3262.451,E2 -3262.451} C_VEL
LIN {X 0,Y 552.148,Z 506.515,A -85,B 0,C 180,E1 -3265.351,E2 -3265.351} C_VEL
LIN {X 0,Y 552.119,Z 506.519,A -85,B 0,C 180,E1 -3268.098,E2 -3268.098} C_VEL
LIN {X 0,Y 552.106,Z 506.527,A -85,B 0,C 180,E1 -3270.609,E2 -3270.609} C_VEL
LIN {X 0,Y 552.122,Z 506.52,A -85,B 0,C 180,E1 -3273.185,E2 -3273.185} C_VEL
LIN {X 0,Y 552.107,Z 506.519,A -85,B 0,C 180,E1 -3275.842,E2 -3275.842} C_VEL
LIN {X 0,Y 552.119,Z 506.523,A -85,B 0,C 180,E1 -3279.062,E2 -3279.062} C_VEL
LIN {X 0,Y 552.133,Z 506.517,A -85,B 0,C 180,E1 -3281.445,E2 -3281.445} C_VEL
LIN {X 0,Y 552.089,Z 506.526,A -85,B 0,C 180,E1 -3284.532,E2 -3284.532} C_VEL
LIN {X 0,Y 552.126,Z 506.517,A -85,B 0,C 180,E1 -3287.585,E2 -3287.585} C_VEL
LIN {X 0,Y 552.13,Z 506.519,A -85,B 0,C 180,E1 -3290.474,E2 -3290.474} C_VEL
LIN {X 0,Y 552.108,Z 506.523,A -85,B 0,C 180,E1 -3293.317,E2 -3293.317} C_VEL
LIN {X 0,Y 552.125,Z 506.518,A -85,B 0,C 180,E1 -3295.94,E2 -3295.94} C_VEL
LIN {X 0,Y 552.116,Z 506.524,A -85,B 0,C 180,E1 -3298.541,E2 -3298.541} C_VEL
LIN {X 0,Y 552.153,Z 506.687,A -85,B 0,C 180,E1 -3301.355,E2 -3301.355} C_VEL
LIN {X 0,Y 553.686,Z 514.988,A -85,B 0,C 180,E1 -3302.687,E2 -3302.687} C_VEL
LIN {X 0,Y 553.492,Z 530.984,A -85,B 0,C 180,E1 -3305.027,E2 -3305.027} C_VEL
LIN {X 0,Y 553.284,Z 549.865,A -85,B 0,C 180,E1 -3307.749,E2 -3307.749} C_VEL
LIN {X 0,Y 552.96,Z 568.532,A -85,B 0,C 180,E1 -3310.418,E2 -3310.418} C_VEL
LIN {X 0,Y 552.612,Z 589.03,A -85,B 0,C 180,E1 -3313.373,E2 -3313.373} C_VEL
LIN {X 0,Y 552.327,Z 608.888,A -85,B 0,C 180,E1 -3316.197,E2 -3316.197} C_VEL
LIN {X 0,Y 552.17,Z 626.649,A -85,B 0,C 180,E1 -3318.664,E2 -3318.664} C_VEL
LIN {X 0,Y 552.764,Z 634.003,A -85,B 0,C 180,E1 -3318.798,E2 -3318.798} C_VEL
LIN {X 0,Y 552.632,Z 704.153,A -85,B 0,C 180,E1 -3319.721,E2 -3319.721} C_VEL
LIN {X 0,Y 552.541,Z 713.426,A -85,B 0,C 180,E1 -3319.928,E2 -3319.928} C_VEL
LIN {X 0,Y 552.514,Z 721.9,A -85,B 0,C 180,E1 -3320.205,E2 -3320.205} C_VEL
LIN {X 0,Y 552.434,Z 730.4,A -85,B 0,C 180,E1 -3320.573,E2 -3320.573} C_VEL
LIN {X 0,Y 552.271,Z 738.73,A -85,B 0,C 180,E1 -3321.032,E2 -3321.032} C_VEL
LIN {X 0,Y 552.173,Z 746.773,A -85,B 0,C 180,E1 -3321.583,E2 -3321.583} C_VEL
LIN {X 0,Y 552.049,Z 755.438,A -85,B 0,C 180,E1 -3322.318,E2 -3322.318} C_VEL
LIN {X 0,Y 551.953,Z 764.434,A -85,B 0,C 180,E1 -3323.3,E2 -3323.3} C_VEL
LIN {X 0,Y 551.917,Z 770.612,A -85,B 0,C 180,E1 -3324.153,E2 -3324.153} C_VEL
LIN {X 0,Y 551.746,Z 774.989,A -85,B 0,C 180,E1 -3324.885,E2 -3324.885} C_VEL
LIN {X 0,Y 551.779,Z 780.149,A -85,B 0,C 180,E1 -3325.983,E2 -3325.983} C_VEL
LIN {X 0,Y 551.731,Z 783.936,A -85,B 0,C 180,E1 -3327.079,E2 -3327.079} C_VEL
LIN {X 0,Y 551.655,Z 785.682,A -85,B 0,C 180,E1 -3327.81,E2 -3327.81} C_VEL
LIN {X 0,Y 551.644,Z 786.933,A -85,B 0,C 180,E1 -3328.54,E2 -3328.54} C_VEL
LIN {X 0,Y 551.639,Z 787.709,A -85,B 0,C 180,E1 -3329.27,E2 -3329.27} C_VEL
LIN {X 0,Y 551.637,Z 788,A -85,B 0,C 180,E1 -3330,E2 -3330} C_VEL
LIN {X 0,Y 551.639,Z 787.709,A -85,B 0,C 180,E1 -3330.73,E2 -3330.73} C_VEL
LIN {X 0,Y 551.644,Z 786.934,A -85,B 0,C 180,E1 -3331.46,E2 -3331.46} C_VEL
LIN {X 0,Y 551.655,Z 785.684,A -85,B 0,C 180,E1 -3332.19,E2 -3332.19} C_VEL
LIN {X 0,Y 551.767,Z 782.789,A -85,B 0,C 180,E1 -3333.286,E2 -3333.286} C_VEL
LIN {X 0,Y 551.773,Z 780.148,A -85,B 0,C 180,E1 -3334.017,E2 -3334.017} C_VEL
LIN {X 0,Y 551.746,Z 774.99,A -85,B 0,C 180,E1 -3335.115,E2 -3335.115} C_VEL
LIN {X 0,Y 551.935,Z 768.441,A -85,B 0,C 180,E1 -3336.179,E2 -3336.179} C_VEL
LIN {X 0,Y 551.996,Z 760.747,A -85,B 0,C 180,E1 -3337.13,E2 -3337.13} C_VEL
LIN {X 0,Y 552.077,Z 753.406,A -85,B 0,C 180,E1 -3337.865,E2 -3337.865} C_VEL
LIN {X 0,Y 552.195,Z 745.544,A -85,B 0,C 180,E1 -3338.508,E2 -3338.508} C_VEL
LIN {X 0,Y 552.3,Z 737.232,A -85,B 0,C 180,E1 -3339.06,E2 -3339.06} C_VEL
LIN {X 0,Y 552.459,Z 726.618,A -85,B 0,C 180,E1 -3339.611,E2 -3339.611} C_VEL
LIN {X 0,Y 552.548,Z 715.087,A -85,B 0,C 180,E1 -3340.026,E2 -3340.026} C_VEL
LIN {X 0,Y 552.587,Z 705.457,A -85,B 0,C 180,E1 -3340.256,E2 -3340.256} C_VEL
LIN {X 0,Y 552.707,Z 673.251,A -85,B 0,C 180,E1 -3340.694,E2 -3340.694} C_VEL
LIN {X 0,Y 552.644,Z 630.705,A -85,B 0,C 180,E1 -3341.247,E2 -3341.247} C_VEL
LIN {X 0,Y 552.155,Z 626.694,A -85,B 0,C 180,E1 -3341.328,E2 -3341.328} C_VEL
LIN {X 0,Y 552.355,Z 607.565,A -85,B 0,C 180,E1 -3343.989,E2 -3343.989} C_VEL
LIN {X 0,Y 552.634,Z 586.383,A -85,B 0,C 180,E1 -3347.007,E2 -3347.007} C_VEL
LIN {X 0,Y 553.033,Z 566.465,A -85,B 0,C 180,E1 -3349.882,E2 -3349.882} C_VEL
LIN {X 0,Y 553.249,Z 546.942,A -85,B 0,C 180,E1 -3352.598,E2 -3352.598} C_VEL
LIN {X 0,Y 553.365,Z 526.87,A -85,B 0,C 180,E1 -3355.381,E2 -3355.381} C_VEL
LIN {X 0,Y 553.353,Z 512.661,A -85,B 0,C 180,E1 -3357.412,E2 -3357.412} C_VEL
LIN {X 0,Y 552.163,Z 506.649,A -85,B 0,C 180,E1 -3358.361,E2 -3358.361} C_VEL
LIN {X 0,Y 552.133,Z 506.52,A -85,B 0,C 180,E1 -3361.479,E2 -3361.479} C_VEL
LIN {X 0,Y 552.131,Z 506.518,A -85,B 0,C 180,E1 -3364.17,E2 -3364.17} C_VEL
LIN {X 0,Y 552.106,Z 506.526,A -85,B 0,C 180,E1 -3366.746,E2 -3366.746} C_VEL
LIN {X 0,Y 552.13,Z 506.518,A -85,B 0,C 180,E1 -3369.526,E2 -3369.526} C_VEL
LIN {X 0,Y 552.126,Z 506.519,A -85,B 0,C 180,E1 -3372.425,E2 -3372.425} C_VEL
LIN {X 0,Y 552.093,Z 506.523,A -85,B 0,C 180,E1 -3375.562,E2 -3375.562} C_VEL
LIN {X 0,Y 552.133,Z 506.52,A -85,B 0,C 180,E1 -3378.675,E2 -3378.675} C_VEL
LIN {X 0,Y 552.114,Z 506.521,A -85,B 0,C 180,E1 -3381.411,E2 -3381.411} C_VEL
LIN {X 0,Y 552.107,Z 506.519,A -85,B 0,C 180,E1 -3384.158,E2 -3384.158} C_VEL
LIN {X 0,Y 552.121,Z 506.526,A -85,B 0,C 180,E1 -3386.815,E2 -3386.815} C_VEL
LIN {X 0,Y 552.106,Z 506.522,A -85,B 0,C 180,E1 -3389.391,E2 -3389.391} C_VEL
LIN {X 0,Y 552.119,Z 506.518,A -85,B 0,C 180,E1 -3391.902,E2 -3391.902} C_VEL
LIN {X 0,Y 552.153,Z 506.518,A -85,B 0,C 180,E1 -3394.647,E2 -3394.647} C_VEL
LIN {X 0,Y 552.087,Z 506.523,A -85,B 0,C 180,E1 -3397.549,E2 -3397.549} C_VEL
LIN {X 0,Y 552.139,Z 506.517,A -85,B 0,C 180,E1 -3400.373,E2 -3400.373} C_VEL
LIN {X 0,Y 552.148,Z 506.523,A -85,B 0,C 180,E1 -3402.977,E2 -3402.977} C_VEL
LIN {X 0,Y 552.127,Z 506.517,A -85,B 0,C 180,E1 -3406.004,E2 -3406.004} C_VEL
LIN {X 0,Y 552.169,Z 506.52,A -85,B 0,C 180,E1 -3408.994,E2 -3408.994} C_VEL
LIN {X 0,Y 552.157,Z 506.514,A -85,B 0,C 180,E1 -3411.952,E2 -3411.952} C_VEL
LIN {X 0,Y 552.229,Z 506.514,A -85,B 0,C 180,E1 -3414.889,E2 -3414.889} C_VEL
LIN {X 0,Y 552.215,Z 506.507,A -85,B 0,C 180,E1 -3417.812,E2 -3417.812} C_VEL
LIN {X 0,Y 552.239,Z 506.512,A -85,B 0,C 180,E1 -3420.729,E2 -3420.729} C_VEL
LIN {X 0,Y 552.204,Z 506.516,A -85,B 0,C 180,E1 -3422.918,E2 -3422.918} C_VEL
LIN {X 0,Y 552.2,Z 506.511,A -85,B 0,C 180,E1 -3425.844,E2 -3425.844} C_VEL
LIN {X 0,Y 552.192,Z 506.688,A -85,B 0,C 180,E1 -3427.625,E2 -3427.625} C_VEL
LIN {X 0,Y 552.381,Z 507.676,A -85,B 0,C 180,E1 -3427.738,E2 -3427.738} C_VEL
LIN {X 0,Y 553.214,Z 510.737,A -85,B 0,C 180,E1 -3427.81,E2 -3427.81} C_VEL
LIN {X 0,Y 553.109,Z 535.056,A -85,B 0,C 180,E1 -3428.15,E2 -3428.15} C_VEL
LIN {X 0,Y 552.986,Z 547.888,A -85,B 0,C 180,E1 -3428.474,E2 -3428.474} C_VEL
LIN {X 0,Y 552.808,Z 560.969,A -85,B 0,C 180,E1 -3428.96,E2 -3428.96} C_VEL
LIN {X 0,Y 552.681,Z 571.931,A -85,B 0,C 180,E1 -3429.516,E2 -3429.516} C_VEL
LIN {X 0,Y 552.496,Z 580.898,A -85,B 0,C 180,E1 -3430.074,E2 -3430.074} C_VEL
LIN {X 0,Y 552.343,Z 589.591,A -85,B 0,C 180,E1 -3430.725,E2 -3430.725} C_VEL
LIN {X 0,Y 552.18,Z 597.978,A -85,B 0,C 180,E1 -3431.475,E2 -3431.475} C_VEL
LIN {X 0,Y 552.073,Z 605.807,A -85,B 0,C 180,E1 -3432.312,E2 -3432.312} C_VEL
LIN {X 0,Y 551.943,Z 611.812,A -85,B 0,C 180,E1 -3433.063,E2 -3433.063} C_VEL
LIN {X 0,Y 551.861,Z 618.134,A -85,B 0,C 180,E1 -3434.003,E2 -3434.003} C_VEL
LIN {X 0,Y 551.833,Z 622.481,A -85,B 0,C 180,E1 -3434.757,E2 -3434.757} C_VEL
LIN {X 0,Y 551.756,Z 627.766,A -85,B 0,C 180,E1 -3435.894,E2 -3435.894} C_VEL
LIN {X 0,Y 551.724,Z 631.861,A -85,B 0,C 180,E1 -3437.037,E2 -3437.037} C_VEL
LIN {X 0,Y 551.686,Z 634.053,A -85,B 0,C 180,E1 -3437.803,E2 -3437.803} C_VEL
LIN {X 0,Y 551.652,Z 635.668,A -85,B 0,C 180,E1 -3438.572,E2 -3438.572} C_VEL
LIN {X 0,Y 551.67,Z 637.027,A -85,B 0,C 180,E1 -3439.49,E2 -3439.49} C_VEL
LIN {X 0,Y 551.634,Z 637.657,A -85,B 0,C 180,E1 -3440.12,E2 -3440.12} C_VEL
LIN {X 0,Y 551.636,Z 637.975,A -85,B 0,C 180,E1 -3440.9,E2 -3440.9} C_VEL
LIN {X 0,Y 551.636,Z 637.192,A -85,B 0,C 180,E1 -3442.471,E2 -3442.471} C_VEL
LIN {X 0,Y 551.655,Z 635.785,A -85,B 0,C 180,E1 -3443.473,E2 -3443.473} C_VEL
LIN {X 0,Y 551.719,Z 633.625,A -85,B 0,C 180,E1 -3444.457,E2 -3444.457} C_VEL
LIN {X 0,Y 551.741,Z 632.384,A -85,B 0,C 180,E1 -3444.875,E2 -3444.875} C_VEL
LIN {X 0,Y 551.052,Z 630.623,A -85,B 0,C 180,E1 -3445.456,E2 -3445.456} C_VEL
LIN {X 0,Y 548.17,Z 627.208,A -85,B 0,C 180,E1 -3446.384,E2 -3446.384} C_VEL
LIN {X 0,Y 545.355,Z 623.143,A -85,B 0,C 180,E1 -3447.288,E2 -3447.288} C_VEL
LIN {X 0,Y 544.775,Z 620.201,A -85,B 0,C 180,E1 -3447.825,E2 -3447.825} C_VEL
LIN {X 0,Y 544.883,Z 614.77,A -85,B 0,C 180,E1 -3448.711,E2 -3448.711} C_VEL
LIN {X 0,Y 545.008,Z 606.962,A -85,B 0,C 180,E1 -3449.767,E2 -3449.767} C_VEL
LIN {X 0,Y 545.189,Z 598.622,A -85,B 0,C 180,E1 -3450.686,E2 -3450.686} C_VEL
LIN {X 0,Y 545.308,Z 591.501,A -85,B 0,C 180,E1 -3451.357,E2 -3451.357} C_VEL
LIN {X 0,Y 545.499,Z 581.964,A -85,B 0,C 180,E1 -3452.104,E2 -3452.104} C_VEL
LIN {X 0,Y 545.698,Z 573.77,A -85,B 0,C 180,E1 -3452.637,E2 -3452.637} C_VEL
LIN {X 0,Y 545.842,Z 565.187,A -85,B 0,C 180,E1 -3453.103,E2 -3453.103} C_VEL
LIN {X 0,Y 546.007,Z 555.007,A -85,B 0,C 180,E1 -3453.542,E2 -3453.542} C_VEL
LIN {X 0,Y 546.12,Z 543.708,A -85,B 0,C 180,E1 -3453.903,E2 -3453.903} C_VEL
LIN {X 0,Y 546.206,Z 532.49,A -85,B 0,C 180,E1 -3454.148,E2 -3454.148} C_VEL
LIN {X 0,Y 546.178,Z 511.224,A -85,B 0,C 180,E1 -3454.441,E2 -3454.441} C_VEL
LIN {X 0,Y 545.264,Z 508.162,A -85,B 0,C 180,E1 -3454.534,E2 -3454.534} C_VEL
LIN {X 0,Y 545.134,Z 507.436,A -85,B 0,C 180,E1 -3454.672,E2 -3454.672} C_VEL
LIN {X 0,Y 545.035,Z 507.409,A -85,B 0,C 180,E1 -3457.305,E2 -3457.305} C_VEL
LIN {X 0,Y 545.071,Z 507.397,A -85,B 0,C 180,E1 -3460.143,E2 -3460.143} C_VEL
LIN {X 0,Y 545.083,Z 507.4,A -85,B 0,C 180,E1 -3463.107,E2 -3463.107} C_VEL
LIN {X 0,Y 545.064,Z 507.396,A -85,B 0,C 180,E1 -3466.225,E2 -3466.225} C_VEL
LIN {X 0,Y 545.1,Z 507.394,A -85,B 0,C 180,E1 -3468.888,E2 -3468.888} C_VEL
LIN {X 0,Y 545.053,Z 507.402,A -85,B 0,C 180,E1 -3471.764,E2 -3471.764} C_VEL
LIN {X 0,Y 545.036,Z 507.4,A -85,B 0,C 180,E1 -3474.533,E2 -3474.533} C_VEL
LIN {X 0,Y 545.081,Z 507.4,A -85,B 0,C 180,E1 -3477.213,E2 -3477.213} C_VEL
LIN {X 0,Y 545.066,Z 507.401,A -85,B 0,C 180,E1 -3479.811,E2 -3479.811} C_VEL
LIN {X 0,Y 545.096,Z 507.392,A -85,B 0,C 180,E1 -3482.345,E2 -3482.345} C_VEL
LIN {X 0,Y 545.12,Z 507.39,A -85,B 0,C 180,E1 -3484.821,E2 -3484.821} C_VEL
LIN {X 0,Y 545.039,Z 507.404,A -85,B 0,C 180,E1 -3487.243,E2 -3487.243} C_VEL
LIN {X 0,Y 545.12,Z 507.389,A -85,B 0,C 180,E1 -3490.415,E2 -3490.415} C_VEL
LIN {X 0,Y 545.07,Z 507.404,A -85,B 0,C 180,E1 -3493.522,E2 -3493.522} C_VEL
LIN {X 0,Y 545.1,Z 507.398,A -85,B 0,C 180,E1 -3495.82,E2 -3495.82} C_VEL
LIN {X 0,Y 545.122,Z 507.389,A -85,B 0,C 180,E1 -3498.85,E2 -3498.85} C_VEL
LIN {X 0,Y 545.133,Z 507.395,A -85,B 0,C 180,E1 -3501.847,E2 -3501.847} C_VEL
LIN {X 0,Y 545.202,Z 507.379,A -85,B 0,C 180,E1 -3504.823,E2 -3504.823} C_VEL
LIN {X 0,Y 545.2,Z 507.388,A -85,B 0,C 180,E1 -3507.784,E2 -3507.784} C_VEL
LIN {X 0,Y 545.215,Z 507.377,A -85,B 0,C 180,E1 -3510.739,E2 -3510.739} C_VEL
LIN {X 0,Y 545.174,Z 507.383,A -85,B 0,C 180,E1 -3512.956,E2 -3512.956} C_VEL
LIN {X 0,Y 545.166,Z 507.391,A -85,B 0,C 180,E1 -3515.919,E2 -3515.919} C_VEL
LIN {X 0,Y 545.113,Z 507.39,A -85,B 0,C 180,E1 -3518.9,E2 -3518.9} C_VEL
LIN {X 0,Y 545.14,Z 507.396,A -85,B 0,C 180,E1 -3521.904,E2 -3521.904} C_VEL
LIN {X 0,Y 545.09,Z 507.393,A -85,B 0,C 180,E1 -3524.943,E2 -3524.943} C_VEL
LIN {X 0,Y 545.084,Z 507.401,A -85,B 0,C 180,E1 -3528.025,E2 -3528.025} C_VEL
LIN {X 0,Y 545.098,Z 507.395,A -85,B 0,C 180,E1 -3530.372,E2 -3530.372} C_VEL
LIN {X 0,Y 545.082,Z 507.398,A -85,B 0,C 180,E1 -3533.559,E2 -3533.559} C_VEL
LIN {X 0,Y 545.082,Z 507.403,A -85,B 0,C 180,E1 -3536,E2 -3536} C_VEL
LIN {X 0,Y 545.091,Z 507.393,A -85,B 0,C 180,E1 -3538.747,E2 -3538.747} C_VEL
LIN {X 0,Y 545.059,Z 507.401,A -85,B 0,C 180,E1 -3541.678,E2 -3541.678} C_VEL
LIN {X 0,Y 545.062,Z 507.398,A -85,B 0,C 180,E1 -3544.564,E2 -3544.564} C_VEL
LIN {X 0,Y 545.036,Z 507.4,A -85,B 0,C 180,E1 -3547.303,E2 -3547.303} C_VEL
LIN {X 0,Y 545.092,Z 507.402,A -85,B 0,C 180,E1 -3550.139,E2 -3550.139} C_VEL
LIN {X 0,Y 545.085,Z 507.393,A -85,B 0,C 180,E1 -3553.105,E2 -3553.105} C_VEL
LIN {X 0,Y 545.064,Z 507.404,A -85,B 0,C 180,E1 -3556.223,E2 -3556.223} C_VEL
LIN {X 0,Y 545.094,Z 507.393,A -85,B 0,C 180,E1 -3558.886,E2 -3558.886} C_VEL
LIN {X 0,Y 545.05,Z 507.401,A -85,B 0,C 180,E1 -3561.762,E2 -3561.762} C_VEL
LIN {X 0,Y 545.061,Z 507.401,A -85,B 0,C 180,E1 -3564.533,E2 -3564.533} C_VEL
LIN {X 0,Y 545.077,Z 507.394,A -85,B 0,C 180,E1 -3567.212,E2 -3567.212} C_VEL
LIN {X 0,Y 545.096,Z 507.395,A -85,B 0,C 180,E1 -3569.812,E2 -3569.812} C_VEL
LIN {X 0,Y 545.095,Z 507.394,A -85,B 0,C 180,E1 -3572.824,E2 -3572.824} C_VEL
LIN {X 0,Y 545.045,Z 507.4,A -85,B 0,C 180,E1 -3575.63,E2 -3575.63} C_VEL
LIN {X 0,Y 545.062,Z 507.399,A -85,B 0,C 180,E1 -3578.836,E2 -3578.836} C_VEL
LIN {X 0,Y 545.077,Z 507.395,A -85,B 0,C 180,E1 -3581.195,E2 -3581.195} C_VEL
LIN {X 0,Y 545.068,Z 507.396,A -85,B 0,C 180,E1 -3583.521,E2 -3583.521} C_VEL
LIN {X 0,Y 545.087,Z 507.395,A -85,B 0,C 180,E1 -3585.819,E2 -3585.819} C_VEL
LIN {X 0,Y 545.109,Z 507.393,A -85,B 0,C 180,E1 -3588.849,E2 -3588.849} C_VEL
LIN {X 0,Y 545.126,Z 507.39,A -85,B 0,C 180,E1 -3591.847,E2 -3591.847} C_VEL
LIN {X 0,Y 545.2,Z 507.383,A -85,B 0,C 180,E1 -3594.823,E2 -3594.823} C_VEL
LIN {X 0,Y 545.187,Z 507.382,A -85,B 0,C 180,E1 -3597.783,E2 -3597.783} C_VEL
LIN {X 0,Y 545.207,Z 507.384,A -85,B 0,C 180,E1 -3600.738,E2 -3600.738} C_VEL
LIN {X 0,Y 545.168,Z 507.386,A -85,B 0,C 180,E1 -3602.956,E2 -3602.956} C_VEL
LIN {X 0,Y 545.163,Z 507.385,A -85,B 0,C 180,E1 -3605.919,E2 -3605.919} C_VEL
LIN {X 0,Y 545.119,Z 507.394,A -85,B 0,C 180,E1 -3608.9,E2 -3608.9} C_VEL
LIN {X 0,Y 545.125,Z 507.389,A -85,B 0,C 180,E1 -3611.904,E2 -3611.904} C_VEL
LIN {X 0,Y 545.076,Z 507.399,A -85,B 0,C 180,E1 -3614.944,E2 -3614.944} C_VEL
LIN {X 0,Y 545.074,Z 507.396,A -85,B 0,C 180,E1 -3618.026,E2 -3618.026} C_VEL
LIN {X 0,Y 545.09,Z 507.398,A -85,B 0,C 180,E1 -3620.372,E2 -3620.372} C_VEL
LIN {X 0,Y 545.082,Z 507.394,A -85,B 0,C 180,E1 -3623.559,E2 -3623.559} C_VEL
LIN {X 0,Y 545.081,Z 507.395,A -85,B 0,C 180,E1 -3626,E2 -3626} C_VEL
LIN {X 0,Y 545.085,Z 507.403,A -85,B 0,C 180,E1 -3628.749,E2 -3628.749} C_VEL
LIN {X 0,Y 545.07,Z 507.395,A -85,B 0,C 180,E1 -3631.683,E2 -3631.683} C_VEL
LIN {X 0,Y 545.078,Z 507.401,A -85,B 0,C 180,E1 -3634.563,E2 -3634.563} C_VEL
LIN {X 0,Y 545.032,Z 507.402,A -85,B 0,C 180,E1 -3637.304,E2 -3637.304} C_VEL
LIN {X 0,Y 545.068,Z 507.397,A -85,B 0,C 180,E1 -3640.142,E2 -3640.142} C_VEL
LIN {X 0,Y 545.072,Z 507.401,A -85,B 0,C 180,E1 -3643.107,E2 -3643.107} C_VEL
LIN {X 0,Y 545.059,Z 507.398,A -85,B 0,C 180,E1 -3646.225,E2 -3646.225} C_VEL
LIN {X 0,Y 545.093,Z 507.403,A -85,B 0,C 180,E1 -3648.888,E2 -3648.888} C_VEL
LIN {X 0,Y 545.05,Z 507.398,A -85,B 0,C 180,E1 -3651.764,E2 -3651.764} C_VEL
LIN {X 0,Y 545.049,Z 507.403,A -85,B 0,C 180,E1 -3654.533,E2 -3654.533} C_VEL
LIN {X 0,Y 545.079,Z 507.403,A -85,B 0,C 180,E1 -3657.213,E2 -3657.213} C_VEL
LIN {X 0,Y 545.064,Z 507.401,A -85,B 0,C 180,E1 -3659.811,E2 -3659.811} C_VEL
LIN {X 0,Y 545.108,Z 507.533,A -85,B 0,C 180,E1 -3661.158,E2 -3661.158} C_VEL
LIN {X 0,Y 546.707,Z 515.633,A -85,B 0,C 180,E1 -3662.499,E2 -3662.499} C_VEL
LIN {X 0,Y 546.601,Z 529.073,A -85,B 0,C 180,E1 -3664.495,E2 -3664.495} C_VEL
LIN {X 0,Y 546.317,Z 548.244,A -85,B 0,C 180,E1 -3667.299,E2 -3667.299} C_VEL
LIN {X 0,Y 545.953,Z 568.444,A -85,B 0,C 180,E1 -3670.223,E2 -3670.223} C_VEL
LIN {X 0,Y 545.744,Z 584.45,A -85,B 0,C 180,E1 -3672.489,E2 -3672.489} C_VEL
LIN {X 0,Y 545.407,Z 606.385,A -85,B 0,C 180,E1 -3675.659,E2 -3675.659} C_VEL
LIN {X 0,Y 545.144,Z 626.618,A -85,B 0,C 180,E1 -3678.513,E2 -3678.513} C_VEL
LIN {X 0,Y 545.748,Z 631.939,A -85,B 0,C 180,E1 -3678.625,E2 -3678.625} C_VEL
LIN {X 0,Y 545.669,Z 704.153,A -85,B 0,C 180,E1 -3679.589,E2 -3679.589} C_VEL
LIN {X 0,Y 545.56,Z 713.426,A -85,B 0,C 180,E1 -3679.798,E2 -3679.798} C_VEL
LIN {X 0,Y 545.533,Z 721.899,A -85,B 0,C 180,E1 -3680.078,E2 -3680.078} C_VEL
LIN {X 0,Y 545.438,Z 730.398,A -85,B 0,C 180,E1 -3680.451,E2 -3680.451} C_VEL
LIN {X 0,Y 545.25,Z 738.728,A -85,B 0,C 180,E1 -3680.915,E2 -3680.915} C_VEL
LIN {X 0,Y 545.158,Z 746.771,A -85,B 0,C 180,E1 -3681.474,E2 -3681.474} C_VEL
LIN {X 0,Y 545.009,Z 755.439,A -85,B 0,C 180,E1 -3682.218,E2 -3682.218} C_VEL
LIN {X 0,Y 544.902,Z 764.083,A -85,B 0,C 180,E1 -3683.167,E2 -3683.167} C_VEL
LIN {X 0,Y 544.843,Z 770.611,A -85,B 0,C 180,E1 -3684.077,E2 -3684.077} C_VEL
LIN {X 0,Y 544.673,Z 774.989,A -85,B 0,C 180,E1 -3684.818,E2 -3684.818} C_VEL
LIN {X 0,Y 544.702,Z 780.149,A -85,B 0,C 180,E1 -3685.931,E2 -3685.931} C_VEL
LIN {X 0,Y 544.66,Z 783.936,A -85,B 0,C 180,E1 -3687.041,E2 -3687.041} C_VEL
LIN {X 0,Y 544.57,Z 785.682,A -85,B 0,C 180,E1 -3687.781,E2 -3687.781} C_VEL
LIN {X 0,Y 544.545,Z 786.932,A -85,B 0,C 180,E1 -3688.521,E2 -3688.521} C_VEL
LIN {X 0,Y 544.54,Z 787.708,A -85,B 0,C 180,E1 -3689.26,E2 -3689.26} C_VEL
LIN {X 0,Y 544.538,Z 788,A -85,B 0,C 180,E1 -3690,E2 -3690} C_VEL
LIN {X 0,Y 544.54,Z 787.709,A -85,B 0,C 180,E1 -3690.739,E2 -3690.739} C_VEL
LIN {X 0,Y 544.545,Z 786.933,A -85,B 0,C 180,E1 -3691.479,E2 -3691.479} C_VEL
LIN {X 0,Y 544.57,Z 785.684,A -85,B 0,C 180,E1 -3692.219,E2 -3692.219} C_VEL
LIN {X 0,Y 544.695,Z 782.789,A -85,B 0,C 180,E1 -3693.328,E2 -3693.328} C_VEL
LIN {X 0,Y 544.697,Z 780.148,A -85,B 0,C 180,E1 -3694.069,E2 -3694.069} C_VEL
LIN {X 0,Y 544.673,Z 774.991,A -85,B 0,C 180,E1 -3695.182,E2 -3695.182} C_VEL
LIN {X 0,Y 544.86,Z 768.962,A -85,B 0,C 180,E1 -3696.183,E2 -3696.183} C_VEL
LIN {X 0,Y 544.944,Z 760.746,A -85,B 0,C 180,E1 -3697.223,E2 -3697.223} C_VEL
LIN {X 0,Y 545.037,Z 753.404,A -85,B 0,C 180,E1 -3697.968,E2 -3697.968} C_VEL
LIN {X 0,Y 545.163,Z 745.542,A -85,B 0,C 180,E1 -3698.619,E2 -3698.619} C_VEL
LIN {X 0,Y 545.284,Z 737.23,A -85,B 0,C 180,E1 -3699.177,E2 -3699.177} C_VEL
LIN {X 0,Y 545.451,Z 726.617,A -85,B 0,C 180,E1 -3699.736,E2 -3699.736} C_VEL
LIN {X 0,Y 545.567,Z 715.087,A -85,B 0,C 180,E1 -3700.155,E2 -3700.155} C_VEL
LIN {X 0,Y 545.622,Z 705.456,A -85,B 0,C 180,E1 -3700.389,E2 -3700.389} C_VEL
LIN {X 0,Y 545.74,Z 673.251,A -85,B 0,C 180,E1 -3700.832,E2 -3700.832} C_VEL
LIN {X 0,Y 545.736,Z 631.584,A -85,B 0,C 180,E1 -3701.38,E2 -3701.38} C_VEL
LIN {X 0,Y 545.139,Z 626.607,A -85,B 0,C 180,E1 -3701.484,E2 -3701.484} C_VEL
LIN {X 0,Y 545.408,Z 606.4,A -85,B 0,C 180,E1 -3704.339,E2 -3704.339} C_VEL
LIN {X 0,Y 545.742,Z 584.454,A -85,B 0,C 180,E1 -3707.51,E2 -3707.51} C_VEL
LIN {X 0,Y 545.958,Z 568.228,A -85,B 0,C 180,E1 -3709.781,E2 -3709.781} C_VEL
LIN {X 0,Y 546.197,Z 547.173,A -85,B 0,C 180,E1 -3712.706,E2 -3712.706} C_VEL
LIN {X 0,Y 546.344,Z 528.694,A -85,B 0,C 180,E1 -3715.309,E2 -3715.309} C_VEL
LIN {X 0,Y 546.384,Z 514.036,A -85,B 0,C 180,E1 -3717.436,E2 -3717.436} C_VEL
LIN {X 0,Y 545.143,Z 507.683,A -85,B 0,C 180,E1 -3718.437,E2 -3718.437} C_VEL
LIN {X 0,Y 545.093,Z 507.4,A -85,B 0,C 180,E1 -3718.749,E2 -3718.749} C_VEL
LIN {X 0,Y 545.069,Z 507.398,A -85,B 0,C 180,E1 -3721.913,E2 -3721.913} C_VEL
LIN {X 0,Y 545.073,Z 507.401,A -85,B 0,C 180,E1 -3724.563,E2 -3724.563} C_VEL
LIN {X 0,Y 545.035,Z 507.405,A -85,B 0,C 180,E1 -3727.303,E2 -3727.303} C_VEL
LIN {X 0,Y 545.07,Z 507.396,A -85,B 0,C 180,E1 -3730.141,E2 -3730.141} C_VEL
LIN {X 0,Y 545.083,Z 507.402,A -85,B 0,C 180,E1 -3733.105,E2 -3733.105} C_VEL
LIN {X 0,Y 545.058,Z 507.398,A -85,B 0,C 180,E1 -3736.224,E2 -3736.224} C_VEL
LIN {X 0,Y 545.094,Z 507.401,A -85,B 0,C 180,E1 -3738.887,E2 -3738.887} C_VEL
LIN {X 0,Y 545.047,Z 507.399,A -85,B 0,C 180,E1 -3741.762,E2 -3741.762} C_VEL
LIN {X 0,Y 545.059,Z 507.4,A -85,B 0,C 180,E1 -3744.533,E2 -3744.533} C_VEL
LIN {X 0,Y 545.074,Z 507.4,A -85,B 0,C 180,E1 -3747.212,E2 -3747.212} C_VEL
LIN {X 0,Y 545.093,Z 507.393,A -85,B 0,C 180,E1 -3749.812,E2 -3749.812} C_VEL
LIN {X 0,Y 545.094,Z 507.402,A -85,B 0,C 180,E1 -3752.824,E2 -3752.824} C_VEL
LIN {X 0,Y 545.048,Z 507.399,A -85,B 0,C 180,E1 -3755.631,E2 -3755.631} C_VEL
LIN {X 0,Y 545.061,Z 507.406,A -85,B 0,C 180,E1 -3758.837,E2 -3758.837} C_VEL
LIN {X 0,Y 545.081,Z 507.399,A -85,B 0,C 180,E1 -3761.196,E2 -3761.196} C_VEL
LIN {X 0,Y 545.068,Z 507.398,A -85,B 0,C 180,E1 -3763.521,E2 -3763.521} C_VEL
LIN {X 0,Y 545.086,Z 507.394,A -85,B 0,C 180,E1 -3765.82,E2 -3765.82} C_VEL
LIN {X 0,Y 545.123,Z 507.398,A -85,B 0,C 180,E1 -3768.85,E2 -3768.85} C_VEL
LIN {X 0,Y 545.127,Z 507.39,A -85,B 0,C 180,E1 -3771.847,E2 -3771.847} C_VEL
LIN {X 0,Y 545.204,Z 507.388,A -85,B 0,C 180,E1 -3774.823,E2 -3774.823} C_VEL
LIN {X 0,Y 545.187,Z 507.382,A -85,B 0,C 180,E1 -3777.784,E2 -3777.784} C_VEL
LIN {X 0,Y 545.209,Z 507.388,A -85,B 0,C 180,E1 -3780.739,E2 -3780.739} C_VEL
LIN {X 0,Y 545.17,Z 507.392,A -85,B 0,C 180,E1 -3782.956,E2 -3782.956} C_VEL
LIN {X 0,Y 545.171,Z 507.388,A -85,B 0,C 180,E1 -3785.92,E2 -3785.92} C_VEL
LIN {X 0,Y 545.152,Z 507.62,A -85,B 0,C 180,E1 -3787.488,E2 -3787.488} C_VEL
LIN {X 0,Y 545.351,Z 508.498,A -85,B 0,C 180,E1 -3787.587,E2 -3787.587} C_VEL
LIN {X 0,Y 546.259,Z 511.536,A -85,B 0,C 180,E1 -3787.661,E2 -3787.661} C_VEL
LIN {X 0,Y 546.169,Z 536.486,A -85,B 0,C 180,E1 -3788.016,E2 -3788.016} C_VEL
LIN {X 0,Y 546.061,Z 550.126,A -85,B 0,C 180,E1 -3788.372,E2 -3788.372} C_VEL
LIN {X 0,Y 545.865,Z 563.109,A -85,B 0,C 180,E1 -3788.888,E2 -3788.888} C_VEL
LIN {X 0,Y 545.715,Z 573.735,A -85,B 0,C 180,E1 -3789.451,E2 -3789.451} C_VEL
LIN {X 0,Y 545.53,Z 582.407,A -85,B 0,C 180,E1 -3790.016,E2 -3790.016} C_VEL
LIN {X 0,Y 545.327,Z 590.854,A -85,B 0,C 180,E1 -3790.677,E2 -3790.677} C_VEL
LIN {X 0,Y 545.149,Z 598.597,A -85,B 0,C 180,E1 -3791.397,E2 -3791.397} C_VEL
LIN {X 0,Y 545.026,Z 606.655,A -85,B 0,C 180,E1 -3792.285,E2 -3792.285} C_VEL
LIN {X 0,Y 544.829,Z 615.055,A -85,B 0,C 180,E1 -3793.426,E2 -3793.426} C_VEL
LIN {X 0,Y 544.763,Z 622.281,A -85,B 0,C 180,E1 -3794.636,E2 -3794.636} C_VEL
LIN {X 0,Y 544.676,Z 627.359,A -85,B 0,C 180,E1 -3795.722,E2 -3795.722} C_VEL
LIN {X 0,Y 544.638,Z 631.547,A -85,B 0,C 180,E1 -3796.879,E2 -3796.879} C_VEL
LIN {X 0,Y 544.57,Z 634.648,A -85,B 0,C 180,E1 -3798.044,E2 -3798.044} C_VEL
LIN {X 0,Y 544.553,Z 636.206,A -85,B 0,C 180,E1 -3798.824,E2 -3798.824} C_VEL
LIN {X 0,Y 544.565,Z 637.183,A -85,B 0,C 180,E1 -3799.606,E2 -3799.606} C_VEL
LIN {X 0,Y 544.552,Z 637.972,A -85,B 0,C 180,E1 -3801.185,E2 -3801.185} C_VEL
LIN {X 0,Y 544.529,Z 637.645,A -85,B 0,C 180,E1 -3801.981,E2 -3801.981} C_VEL
LIN {X 0,Y 544.57,Z 635.582,A -85,B 0,C 180,E1 -3803.613,E2 -3803.613} C_VEL
LIN {X 0,Y 544.65,Z 632.759,A -85,B 0,C 180,E1 -3804.795,E2 -3804.795} C_VEL
LIN {X 0,Y 544.651,Z 629.98,A -85,B 0,C 180,E1 -3805.685,E2 -3805.685} C_VEL
LIN {X 0,Y 544.704,Z 625.211,A -85,B 0,C 180,E1 -3806.846,E2 -3806.846} C_VEL
LIN {X 0,Y 544.775,Z 620.201,A -85,B 0,C 180,E1 -3807.825,E2 -3807.825} C_VEL
LIN {X 0,Y 544.212,Z 617.153,A -85,B 0,C 180,E1 -3808.353,E2 -3808.353} C_VEL
LIN {X 0,Y 541.49,Z 612.087,A -85,B 0,C 180,E1 -3809.211,E2 -3809.211} C_VEL
LIN {X 0,Y 538.756,Z 606.499,A -85,B 0,C 180,E1 -3810.03,E2 -3810.03} C_VEL
LIN {X 0,Y 538.168,Z 602.559,A -85,B 0,C 180,E1 -3810.494,E2 -3810.494} C_VEL
LIN {X 0,Y 538.377,Z 592.469,A -85,B 0,C 180,E1 -3811.478,E2 -3811.478} C_VEL
LIN {X 0,Y 538.588,Z 583.001,A -85,B 0,C 180,E1 -3812.228,E2 -3812.228} C_VEL
LIN {X 0,Y 538.809,Z 572.808,A -85,B 0,C 180,E1 -3812.884,E2 -3812.884} C_VEL
LIN {X 0,Y 538.954,Z 563.841,A -85,B 0,C 180,E1 -3813.351,E2 -3813.351} C_VEL
LIN {X 0,Y 539.124,Z 553.322,A -85,B 0,C 180,E1 -3813.782,E2 -3813.782} C_VEL
LIN {X 0,Y 539.222,Z 542.487,A -85,B 0,C 180,E1 -3814.109,E2 -3814.109} C_VEL
LIN {X 0,Y 539.303,Z 530.791,A -85,B 0,C 180,E1 -3814.343,E2 -3814.343} C_VEL
LIN {X 0,Y 539.201,Z 512.289,A -85,B 0,C 180,E1 -3814.596,E2 -3814.596} C_VEL
LIN {X 0,Y 538.246,Z 509.158,A -85,B 0,C 180,E1 -3814.684,E2 -3814.684} C_VEL
LIN {X 0,Y 538.111,Z 508.339,A -85,B 0,C 180,E1 -3814.823,E2 -3814.823} C_VEL
LIN {X 0,Y 537.989,Z 508.282,A -85,B 0,C 180,E1 -3817.878,E2 -3817.878} C_VEL
LIN {X 0,Y 538.048,Z 508.274,A -85,B 0,C 180,E1 -3820.776,E2 -3820.776} C_VEL
LIN {X 0,Y 538.026,Z 508.274,A -85,B 0,C 180,E1 -3824.076,E2 -3824.076} C_VEL
LIN {X 0,Y 538.023,Z 508.28,A -85,B 0,C 180,E1 -3827.216,E2 -3827.216} C_VEL
LIN {X 0,Y 538.053,Z 508.27,A -85,B 0,C 180,E1 -3830.207,E2 -3830.207} C_VEL
LIN {X 0,Y 538.023,Z 508.277,A -85,B 0,C 180,E1 -3833.068,E2 -3833.068} C_VEL
LIN {X 0,Y 538.019,Z 508.278,A -85,B 0,C 180,E1 -3835.828,E2 -3835.828} C_VEL
LIN {X 0,Y 538.011,Z 508.275,A -85,B 0,C 180,E1 -3838.5,E2 -3838.5} C_VEL
LIN {X 0,Y 538.061,Z 508.272,A -85,B 0,C 180,E1 -3841.101,E2 -3841.101} C_VEL
LIN {X 0,Y 538.045,Z 508.279,A -85,B 0,C 180,E1 -3843.634,E2 -3843.634} C_VEL
LIN {X 0,Y 538.009,Z 508.277,A -85,B 0,C 180,E1 -3846.123,E2 -3846.123} C_VEL
LIN {X 0,Y 538.041,Z 508.277,A -85,B 0,C 180,E1 -3849.349,E2 -3849.349} C_VEL
LIN {X 0,Y 538.04,Z 508.271,A -85,B 0,C 180,E1 -3852.468,E2 -3852.468} C_VEL
LIN {X 0,Y 538.069,Z 508.278,A -85,B 0,C 180,E1 -3855.631,E2 -3855.631} C_VEL
LIN {X 0,Y 538.082,Z 508.266,A -85,B 0,C 180,E1 -3858.702,E2 -3858.702} C_VEL
LIN {X 0,Y 538.089,Z 508.274,A -85,B 0,C 180,E1 -3861.74,E2 -3861.74} C_VEL
LIN {X 0,Y 538.16,Z 508.256,A -85,B 0,C 180,E1 -3864.755,E2 -3864.755} C_VEL
LIN {X 0,Y 538.172,Z 508.264,A -85,B 0,C 180,E1 -3867.755,E2 -3867.755} C_VEL
LIN {X 0,Y 538.185,Z 508.253,A -85,B 0,C 180,E1 -3870.748,E2 -3870.748} C_VEL
LIN {X 0,Y 538.141,Z 508.259,A -85,B 0,C 180,E1 -3872.994,E2 -3872.994} C_VEL
LIN {X 0,Y 538.118,Z 508.268,A -85,B 0,C 180,E1 -3875.997,E2 -3875.997} C_VEL
LIN {X 0,Y 538.066,Z 508.268,A -85,B 0,C 180,E1 -3879.018,E2 -3879.018} C_VEL
LIN {X 0,Y 538.088,Z 508.271,A -85,B 0,C 180,E1 -3882.062,E2 -3882.062} C_VEL
LIN {X 0,Y 538.05,Z 508.271,A -85,B 0,C 180,E1 -3885.143,E2 -3885.143} C_VEL
LIN {X 0,Y 538.036,Z 508.276,A -85,B 0,C 180,E1 -3888.27,E2 -3888.27} C_VEL
LIN {X 0,Y 538.042,Z 508.271,A -85,B 0,C 180,E1 -3890.651,E2 -3890.651} C_VEL
LIN {X 0,Y 538.006,Z 508.285,A -85,B 0,C 180,E1 -3893.888,E2 -3893.888} C_VEL
LIN {X 0,Y 538.044,Z 508.274,A -85,B 0,C 180,E1 -3896.366,E2 -3896.366} C_VEL
LIN {X 0,Y 538.032,Z 508.272,A -85,B 0,C 180,E1 -3898.933,E2 -3898.933} C_VEL
LIN {X 0,Y 538.012,Z 508.283,A -85,B 0,C 180,E1 -3901.886,E2 -3901.886} C_VEL
LIN {X 0,Y 538.012,Z 508.276,A -85,B 0,C 180,E1 -3904.617,E2 -3904.617} C_VEL
LIN {X 0,Y 538.004,Z 508.276,A -85,B 0,C 180,E1 -3907.169,E2 -3907.169} C_VEL
LIN {X 0,Y 538.054,Z 508.275,A -85,B 0,C 180,E1 -3909.793,E2 -3909.793} C_VEL
LIN {X 0,Y 538.022,Z 508.274,A -85,B 0,C 180,E1 -3912.784,E2 -3912.784} C_VEL
LIN {X 0,Y 538.027,Z 508.279,A -85,B 0,C 180,E1 -3915.924,E2 -3915.924} C_VEL
LIN {X 0,Y 538.048,Z 508.27,A -85,B 0,C 180,E1 -3919.251,E2 -3919.251} C_VEL
LIN {X 0,Y 537.99,Z 508.287,A -85,B 0,C 180,E1 -3922.122,E2 -3922.122} C_VEL
LIN {X 0,Y 538.016,Z 508.275,A -85,B 0,C 180,E1 -3924.916,E2 -3924.916} C_VEL
LIN {X 0,Y 538.026,Z 508.274,A -85,B 0,C 180,E1 -3927.617,E2 -3927.617} C_VEL
LIN {X 0,Y 538.038,Z 508.282,A -85,B 0,C 180,E1 -3930.24,E2 -3930.24} C_VEL
LIN {X 0,Y 538.065,Z 508.27,A -85,B 0,C 180,E1 -3932.796,E2 -3932.796} C_VEL
LIN {X 0,Y 538.043,Z 508.271,A -85,B 0,C 180,E1 -3935.292,E2 -3935.292} C_VEL
LIN {X 0,Y 538.008,Z 508.281,A -85,B 0,C 180,E1 -3938.041,E2 -3938.041} C_VEL
LIN {X 0,Y 538.033,Z 508.273,A -85,B 0,C 180,E1 -3940.94,E2 -3940.94} C_VEL
LIN {X 0,Y 538.019,Z 508.274,A -85,B 0,C 180,E1 -3943.298,E2 -3943.298} C_VEL
LIN {X 0,Y 538.055,Z 508.27,A -85,B 0,C 180,E1 -3945.63,E2 -3945.63} C_VEL
LIN {X 0,Y 538.068,Z 508.272,A -85,B 0,C 180,E1 -3948.701,E2 -3948.701} C_VEL
LIN {X 0,Y 538.082,Z 508.267,A -85,B 0,C 180,E1 -3951.739,E2 -3951.739} C_VEL
LIN {X 0,Y 538.176,Z 508.259,A -85,B 0,C 180,E1 -3954.755,E2 -3954.755} C_VEL
LIN {X 0,Y 538.159,Z 508.257,A -85,B 0,C 180,E1 -3957.754,E2 -3957.754} C_VEL
LIN {X 0,Y 538.177,Z 508.26,A -85,B 0,C 180,E1 -3960.748,E2 -3960.748} C_VEL
LIN {X 0,Y 538.134,Z 508.262,A -85,B 0,C 180,E1 -3962.994,E2 -3962.994} C_VEL
LIN {X 0,Y 538.116,Z 508.264,A -85,B 0,C 180,E1 -3965.997,E2 -3965.997} C_VEL
LIN {X 0,Y 538.068,Z 508.271,A -85,B 0,C 180,E1 -3969.017,E2 -3969.017} C_VEL
LIN {X 0,Y 538.074,Z 508.269,A -85,B 0,C 180,E1 -3972.062,E2 -3972.062} C_VEL
LIN {X 0,Y 538.036,Z 508.274,A -85,B 0,C 180,E1 -3975.144,E2 -3975.144} C_VEL
LIN {X 0,Y 538.026,Z 508.277,A -85,B 0,C 180,E1 -3978.27,E2 -3978.27} C_VEL
LIN {X 0,Y 538.033,Z 508.282,A -85,B 0,C 180,E1 -3980.651,E2 -3980.651} C_VEL
LIN {X 0,Y 538.015,Z 508.274,A -85,B 0,C 180,E1 -3983.888,E2 -3983.888} C_VEL
LIN {X 0,Y 538.042,Z 508.275,A -85,B 0,C 180,E1 -3986.366,E2 -3986.366} C_VEL
LIN {X 0,Y 538.048,Z 508.276,A -85,B 0,C 180,E1 -3988.939,E2 -3988.939} C_VEL
LIN {X 0,Y 538.02,Z 508.274,A -85,B 0,C 180,E1 -3991.891,E2 -3991.891} C_VEL
LIN {X 0,Y 538.028,Z 508.28,A -85,B 0,C 180,E1 -3994.622,E2 -3994.622} C_VEL
LIN {X 0,Y 538.001,Z 508.28,A -85,B 0,C 180,E1 -3997.171,E2 -3997.171} C_VEL
LIN {X 0,Y 538.023,Z 508.273,A -85,B 0,C 180,E1 -3999.797,E2 -3999.797} C_VEL
LIN {X 0,Y 538.013,Z 508.284,A -85,B 0,C 180,E1 -4002.786,E2 -4002.786} C_VEL
LIN {X 0,Y 538.026,Z 508.278,A -85,B 0,C 180,E1 -4005.141,E2 -4005.141} C_VEL
LIN {X 0,Y 538.036,Z 508.273,A -85,B 0,C 180,E1 -4008.228,E2 -4008.228} C_VEL
LIN {X 0,Y 538.012,Z 508.28,A -85,B 0,C 180,E1 -4011.17,E2 -4011.17} C_VEL
LIN {X 0,Y 538.02,Z 508.275,A -85,B 0,C 180,E1 -4014.085,E2 -4014.085} C_VEL
LIN {X 0,Y 538.028,Z 508.281,A -85,B 0,C 180,E1 -4016.728,E2 -4016.728} C_VEL
LIN {X 0,Y 538.024,Z 508.281,A -85,B 0,C 180,E1 -4019.557,E2 -4019.557} C_VEL
LIN {X 0,Y 538.065,Z 508.381,A -85,B 0,C 180,E1 -4020.957,E2 -4020.957} C_VEL
LIN {X 0,Y 539.309,Z 514.494,A -85,B 0,C 180,E1 -4022.023,E2 -4022.023} C_VEL
LIN {X 0,Y 539.875,Z 520.093,A -85,B 0,C 180,E1 -4022.896,E2 -4022.896} C_VEL
LIN {X 0,Y 539.426,Z 542.124,A -85,B 0,C 180,E1 -4026.179,E2 -4026.179} C_VEL
LIN {X 0,Y 539.133,Z 558.46,A -85,B 0,C 180,E1 -4028.593,E2 -4028.593} C_VEL
LIN {X 0,Y 538.829,Z 574.74,A -85,B 0,C 180,E1 -4030.97,E2 -4030.97} C_VEL
LIN {X 0,Y 538.517,Z 595.533,A -85,B 0,C 180,E1 -4033.9,E2 -4033.9} C_VEL
LIN {X 0,Y 538.272,Z 612.859,A -85,B 0,C 180,E1 -4036.408,E2 -4036.408} C_VEL
LIN {X 0,Y 538.12,Z 626.442,A -85,B 0,C 180,E1 -4038.347,E2 -4038.347} C_VEL
LIN {X 0,Y 538.362,Z 629.049,A -85,B 0,C 180,E1 -4038.429,E2 -4038.429} C_VEL
LIN {X 0,Y 538.875,Z 635.733,A -85,B 0,C 180,E1 -4038.529,E2 -4038.529} C_VEL
LIN {X 0,Y 538.709,Z 704.153,A -85,B 0,C 180,E1 -4039.453,E2 -4039.453} C_VEL
LIN {X 0,Y 538.588,Z 713.426,A -85,B 0,C 180,E1 -4039.664,E2 -4039.664} C_VEL
LIN {X 0,Y 538.559,Z 721.898,A -85,B 0,C 180,E1 -4039.948,E2 -4039.948} C_VEL
LIN {X 0,Y 538.433,Z 730.396,A -85,B 0,C 180,E1 -4040.326,E2 -4040.326} C_VEL
LIN {X 0,Y 538.24,Z 738.726,A -85,B 0,C 180,E1 -4040.796,E2 -4040.796} C_VEL
LIN {X 0,Y 538.136,Z 746.768,A -85,B 0,C 180,E1 -4041.362,E2 -4041.362} C_VEL
LIN {X 0,Y 537.97,Z 755.44,A -85,B 0,C 180,E1 -4042.116,E2 -4042.116} C_VEL
LIN {X 0,Y 537.821,Z 763.94,A -85,B 0,C 180,E1 -4043.058,E2 -4043.058} C_VEL
LIN {X 0,Y 537.765,Z 770.611,A -85,B 0,C 180,E1 -4043.999,E2 -4043.999} C_VEL
LIN {X 0,Y 537.605,Z 774.989,A -85,B 0,C 180,E1 -4044.75,E2 -4044.75} C_VEL
LIN {X 0,Y 537.626,Z 780.149,A -85,B 0,C 180,E1 -4045.877,E2 -4045.877} C_VEL
LIN {X 0,Y 537.563,Z 783.937,A -85,B 0,C 180,E1 -4047.002,E2 -4047.002} C_VEL
LIN {X 0,Y 537.489,Z 785.682,A -85,B 0,C 180,E1 -4047.752,E2 -4047.752} C_VEL
LIN {X 0,Y 537.45,Z 786.931,A -85,B 0,C 180,E1 -4048.501,E2 -4048.501} C_VEL
LIN {X 0,Y 537.44,Z 787.707,A -85,B 0,C 180,E1 -4049.251,E2 -4049.251} C_VEL
LIN {X 0,Y 537.439,Z 788,A -85,B 0,C 180,E1 -4050,E2 -4050} C_VEL
LIN {X 0,Y 537.44,Z 787.708,A -85,B 0,C 180,E1 -4050.749,E2 -4050.749} C_VEL
LIN {X 0,Y 537.45,Z 786.932,A -85,B 0,C 180,E1 -4051.499,E2 -4051.499} C_VEL
LIN {X 0,Y 537.489,Z 785.684,A -85,B 0,C 180,E1 -4052.248,E2 -4052.248} C_VEL
LIN {X 0,Y 537.595,Z 782.788,A -85,B 0,C 180,E1 -4053.372,E2 -4053.372} C_VEL
LIN {X 0,Y 537.622,Z 780.149,A -85,B 0,C 180,E1 -4054.123,E2 -4054.123} C_VEL
LIN {X 0,Y 537.605,Z 774.99,A -85,B 0,C 180,E1 -4055.25,E2 -4055.25} C_VEL
LIN {X 0,Y 537.786,Z 769.208,A -85,B 0,C 180,E1 -4056.226,E2 -4056.226} C_VEL
LIN {X 0,Y 537.859,Z 762.439,A -85,B 0,C 180,E1 -4057.13,E2 -4057.13} C_VEL
LIN {X 0,Y 537.992,Z 754.423,A -85,B 0,C 180,E1 -4057.978,E2 -4057.978} C_VEL
LIN {X 0,Y 538.136,Z 746.769,A -85,B 0,C 180,E1 -4058.638,E2 -4058.638} C_VEL
LIN {X 0,Y 538.241,Z 738.728,A -85,B 0,C 180,E1 -4059.204,E2 -4059.204} C_VEL
LIN {X 0,Y 538.419,Z 730.397,A -85,B 0,C 180,E1 -4059.675,E2 -4059.675} C_VEL
LIN {X 0,Y 538.505,Z 721.894,A -85,B 0,C 180,E1 -4060.053,E2 -4060.053} C_VEL
LIN {X 0,Y 538.582,Z 711.76,A -85,B 0,C 180,E1 -4060.383,E2 -4060.383} C_VEL
LIN {X 0,Y 538.787,Z 700.081,A -85,B 0,C 180,E1 -4060.617,E2 -4060.617} C_VEL
LIN {X 0,Y 538.777,Z 632.116,A -85,B 0,C 180,E1 -4061.521,E2 -4061.521} C_VEL
LIN {X 0,Y 538.137,Z 626.611,A -85,B 0,C 180,E1 -4061.636,E2 -4061.636} C_VEL
LIN {X 0,Y 538.397,Z 605.39,A -85,B 0,C 180,E1 -4064.677,E2 -4064.677} C_VEL
LIN {X 0,Y 538.628,Z 588.513,A -85,B 0,C 180,E1 -4067.072,E2 -4067.072} C_VEL
LIN {X 0,Y 538.938,Z 567.035,A -85,B 0,C 180,E1 -4070.042,E2 -4070.042} C_VEL
LIN {X 0,Y 539.143,Z 545.924,A -85,B 0,C 180,E1 -4073.02,E2 -4073.02} C_VEL
LIN {X 0,Y 539.378,Z 527.192,A -85,B 0,C 180,E1 -4075.719,E2 -4075.719} C_VEL
LIN {X 0,Y 539.449,Z 516.069,A -85,B 0,C 180,E1 -4077.36,E2 -4077.36} C_VEL
LIN {X 0,Y 538.088,Z 508.468,A -85,B 0,C 180,E1 -4078.578,E2 -4078.578} C_VEL
LIN {X 0,Y 538.021,Z 508.278,A -85,B 0,C 180,E1 -4081.5,E2 -4081.5} C_VEL
LIN {X 0,Y 538.02,Z 508.276,A -85,B 0,C 180,E1 -4084.172,E2 -4084.172} C_VEL
LIN {X 0,Y 538.003,Z 508.283,A -85,B 0,C 180,E1 -4087.17,E2 -4087.17} C_VEL
LIN {X 0,Y 538.025,Z 508.274,A -85,B 0,C 180,E1 -4089.796,E2 -4089.796} C_VEL
LIN {X 0,Y 538.02,Z 508.281,A -85,B 0,C 180,E1 -4092.785,E2 -4092.785} C_VEL
LIN {X 0,Y 538.022,Z 508.274,A -85,B 0,C 180,E1 -4095.925,E2 -4095.925} C_VEL
LIN {X 0,Y 538.071,Z 508.273,A -85,B 0,C 180,E1 -4099.248,E2 -4099.248} C_VEL
LIN {X 0,Y 537.995,Z 508.278,A -85,B 0,C 180,E1 -4102.123,E2 -4102.123} C_VEL
LIN {X 0,Y 538.015,Z 508.282,A -85,B 0,C 180,E1 -4104.917,E2 -4104.917} C_VEL
LIN {X 0,Y 538.023,Z 508.274,A -85,B 0,C 180,E1 -4107.618,E2 -4107.618} C_VEL
LIN {X 0,Y 538.035,Z 508.273,A -85,B 0,C 180,E1 -4110.24,E2 -4110.24} C_VEL
LIN {X 0,Y 538.063,Z 508.277,A -85,B 0,C 180,E1 -4112.796,E2 -4112.796} C_VEL
LIN {X 0,Y 538.045,Z 508.275,A -85,B 0,C 180,E1 -4115.293,E2 -4115.293} C_VEL
LIN {X 0,Y 538.005,Z 508.277,A -85,B 0,C 180,E1 -4118.042,E2 -4118.042} C_VEL
LIN {X 0,Y 538.036,Z 508.281,A -85,B 0,C 180,E1 -4120.94,E2 -4120.94} C_VEL
LIN {X 0,Y 538.019,Z 508.278,A -85,B 0,C 180,E1 -4123.299,E2 -4123.299} C_VEL
LIN {X 0,Y 538.054,Z 508.271,A -85,B 0,C 180,E1 -4125.631,E2 -4125.631} C_VEL
LIN {X 0,Y 538.08,Z 508.274,A -85,B 0,C 180,E1 -4128.702,E2 -4128.702} C_VEL
LIN {X 0,Y 538.083,Z 508.268,A -85,B 0,C 180,E1 -4131.74,E2 -4131.74} C_VEL
LIN {X 0,Y 538.18,Z 508.263,A -85,B 0,C 180,E1 -4134.755,E2 -4134.755} C_VEL
LIN {X 0,Y 538.159,Z 508.258,A -85,B 0,C 180,E1 -4137.755,E2 -4137.755} C_VEL
LIN {X 0,Y 538.178,Z 508.263,A -85,B 0,C 180,E1 -4140.749,E2 -4140.749} C_VEL
LIN {X 0,Y 538.136,Z 508.268,A -85,B 0,C 180,E1 -4142.995,E2 -4142.995} C_VEL
LIN {X 0,Y 538.125,Z 508.266,A -85,B 0,C 180,E1 -4145.998,E2 -4145.998} C_VEL
LIN {X 0,Y 538.097,Z 508.375,A -85,B 0,C 180,E1 -4147.298,E2 -4147.298} C_VEL
LIN {X 0,Y 538.3,Z 509.416,A -85,B 0,C 180,E1 -4147.437,E2 -4147.437} C_VEL
LIN {X 0,Y 539.253,Z 512.582,A -85,B 0,C 180,E1 -4147.512,E2 -4147.512} C_VEL
LIN {X 0,Y 539.264,Z 537.183,A -85,B 0,C 180,E1 -4147.865,E2 -4147.865} C_VEL
LIN {X 0,Y 539.147,Z 550.765,A -85,B 0,C 180,E1 -4148.218,E2 -4148.218} C_VEL
LIN {X 0,Y 538.963,Z 563.536,A -85,B 0,C 180,E1 -4148.719,E2 -4148.719} C_VEL
LIN {X 0,Y 538.82,Z 574.313,A -85,B 0,C 180,E1 -4149.289,E2 -4149.289} C_VEL
LIN {X 0,Y 538.581,Z 584.377,A -85,B 0,C 180,E1 -4149.957,E2 -4149.957} C_VEL
LIN {X 0,Y 538.363,Z 593.765,A -85,B 0,C 180,E1 -4150.721,E2 -4150.721} C_VEL
LIN {X 0,Y 538.155,Z 603.024,A -85,B 0,C 180,E1 -4151.64,E2 -4151.64} C_VEL
LIN {X 0,Y 537.966,Z 612.568,A -85,B 0,C 180,E1 -4152.832,E2 -4152.832} C_VEL
LIN {X 0,Y 537.804,Z 618.806,A -85,B 0,C 180,E1 -4153.798,E2 -4153.798} C_VEL
LIN {X 0,Y 537.725,Z 623.804,A -85,B 0,C 180,E1 -4154.727,E2 -4154.727} C_VEL
LIN {X 0,Y 537.611,Z 628.971,A -85,B 0,C 180,E1 -4155.934,E2 -4155.934} C_VEL
LIN {X 0,Y 537.578,Z 631.719,A -85,B 0,C 180,E1 -4156.716,E2 -4156.716} C_VEL
LIN {X 0,Y 537.548,Z 633.901,A -85,B 0,C 180,E1 -4157.5,E2 -4157.5} C_VEL
LIN {X 0,Y 537.475,Z 636.909,A -85,B 0,C 180,E1 -4159.081,E2 -4159.081} C_VEL
LIN {X 0,Y 537.453,Z 637.821,A -85,B 0,C 180,E1 -4159.877,E2 -4159.877} C_VEL
LIN {X 0,Y 537.461,Z 638.208,A -85,B 0,C 180,E1 -4161.478,E2 -4161.478} C_VEL
LIN {X 0,Y 537.441,Z 637.752,A -85,B 0,C 180,E1 -4162.286,E2 -4162.286} C_VEL
LIN {X 0,Y 537.502,Z 635.725,A -85,B 0,C 180,E1 -4163.759,E2 -4163.759} C_VEL
LIN {X 0,Y 537.581,Z 632.314,A -85,B 0,C 180,E1 -4165.144,E2 -4165.144} C_VEL
LIN {X 0,Y 537.601,Z 629.607,A -85,B 0,C 180,E1 -4165.973,E2 -4165.973} C_VEL
LIN {X 0,Y 537.676,Z 626.342,A -85,B 0,C 180,E1 -4166.805,E2 -4166.805} C_VEL
LIN {X 0,Y 537.811,Z 620.094,A -85,B 0,C 180,E1 -4168.063,E2 -4168.063} C_VEL
LIN {X 0,Y 537.921,Z 613.388,A -85,B 0,C 180,E1 -4169.123,E2 -4169.123} C_VEL
LIN {X 0,Y 538.043,Z 606.972,A -85,B 0,C 180,E1 -4169.975,E2 -4169.975} C_VEL
LIN {X 0,Y 538.168,Z 602.559,A -85,B 0,C 180,E1 -4170.494,E2 -4170.494} C_VEL
LIN {X 0,Y 537.549,Z 599.844,A -85,B 0,C 180,E1 -4170.798,E2 -4170.798} C_VEL
LIN {X 0,Y 532.123,Z 591.379,A -85,B 0,C 180,E1 -4171.768,E2 -4171.768} C_VEL
LIN {X 0,Y 531.565,Z 588.317,A -85,B 0,C 180,E1 -4172.036,E2 -4172.036} C_VEL
LIN {X 0,Y 531.811,Z 577.414,A -85,B 0,C 180,E1 -4172.808,E2 -4172.808} C_VEL
LIN {X 0,Y 532.061,Z 565.402,A -85,B 0,C 180,E1 -4173.469,E2 -4173.469} C_VEL
LIN {X 0,Y 532.221,Z 554.869,A -85,B 0,C 180,E1 -4173.912,E2 -4173.912} C_VEL
LIN {X 0,Y 532.322,Z 542.964,A -85,B 0,C 180,E1 -4174.275,E2 -4174.275} C_VEL
LIN {X 0,Y 532.389,Z 529.613,A -85,B 0,C 180,E1 -4174.529,E2 -4174.529} C_VEL
LIN {X 0,Y 532.33,Z 513.693,A -85,B 0,C 180,E1 -4174.747,E2 -4174.747} C_VEL
LIN {X 0,Y 531.208,Z 509.925,A -85,B 0,C 180,E1 -4174.858,E2 -4174.858} C_VEL
LIN {X 0,Y 531.044,Z 509.212,A -85,B 0,C 180,E1 -4175.005,E2 -4175.005} C_VEL
LIN {X 0,Y 530.962,Z 509.161,A -85,B 0,C 180,E1 -4177.508,E2 -4177.508} C_VEL
LIN {X 0,Y 530.981,Z 509.152,A -85,B 0,C 180,E1 -4180.433,E2 -4180.433} C_VEL
LIN {X 0,Y 530.967,Z 509.161,A -85,B 0,C 180,E1 -4183.283,E2 -4183.283} C_VEL
LIN {X 0,Y 530.986,Z 509.156,A -85,B 0,C 180,E1 -4185.622,E2 -4185.622} C_VEL
LIN {X 0,Y 531.006,Z 509.148,A -85,B 0,C 180,E1 -4188.567,E2 -4188.567} C_VEL
LIN {X 0,Y 530.968,Z 509.161,A -85,B 0,C 180,E1 -4191.347,E2 -4191.347} C_VEL
LIN {X 0,Y 530.953,Z 509.154,A -85,B 0,C 180,E1 -4194.381,E2 -4194.381} C_VEL
LIN {X 0,Y 530.97,Z 509.156,A -85,B 0,C 180,E1 -4197.135,E2 -4197.135} C_VEL
LIN {X 0,Y 530.971,Z 509.156,A -85,B 0,C 180,E1 -4199.804,E2 -4199.804} C_VEL
LIN {X 0,Y 531.018,Z 509.146,A -85,B 0,C 180,E1 -4202.467,E2 -4202.467} C_VEL
LIN {X 0,Y 531.008,Z 509.149,A -85,B 0,C 180,E1 -4204.943,E2 -4204.943} C_VEL
LIN {X 0,Y 530.974,Z 509.152,A -85,B 0,C 180,E1 -4208.247,E2 -4208.247} C_VEL
LIN {X 0,Y 530.996,Z 509.149,A -85,B 0,C 180,E1 -4210.678,E2 -4210.678} C_VEL
LIN {X 0,Y 530.975,Z 509.153,A -85,B 0,C 180,E1 -4213.071,E2 -4213.071} C_VEL
LIN {X 0,Y 531.024,Z 509.152,A -85,B 0,C 180,E1 -4215.436,E2 -4215.436} C_VEL
LIN {X 0,Y 531.042,Z 509.143,A -85,B 0,C 180,E1 -4218.55,E2 -4218.55} C_VEL
LIN {X 0,Y 531.058,Z 509.15,A -85,B 0,C 180,E1 -4221.63,E2 -4221.63} C_VEL
LIN {X 0,Y 531.119,Z 509.133,A -85,B 0,C 180,E1 -4224.685,E2 -4224.685} C_VEL
LIN {X 0,Y 531.144,Z 509.14,A -85,B 0,C 180,E1 -4227.725,E2 -4227.725} C_VEL
LIN {X 0,Y 531.156,Z 509.129,A -85,B 0,C 180,E1 -4230.758,E2 -4230.758} C_VEL
LIN {X 0,Y 531.108,Z 509.135,A -85,B 0,C 180,E1 -4233.034,E2 -4233.034} C_VEL
LIN {X 0,Y 531.073,Z 509.144,A -85,B 0,C 180,E1 -4236.077,E2 -4236.077} C_VEL
LIN {X 0,Y 531.028,Z 509.145,A -85,B 0,C 180,E1 -4239.138,E2 -4239.138} C_VEL
LIN {X 0,Y 531.046,Z 509.146,A -85,B 0,C 180,E1 -4242.225,E2 -4242.225} C_VEL
LIN {X 0,Y 530.999,Z 509.15,A -85,B 0,C 180,E1 -4245.349,E2 -4245.349} C_VEL
LIN {X 0,Y 530.994,Z 509.15,A -85,B 0,C 180,E1 -4248.521,E2 -4248.521} C_VEL
LIN {X 0,Y 531.003,Z 509.148,A -85,B 0,C 180,E1 -4250.937,E2 -4250.937} C_VEL
LIN {X 0,Y 530.968,Z 509.157,A -85,B 0,C 180,E1 -4254.225,E2 -4254.225} C_VEL
LIN {X 0,Y 531.007,Z 509.148,A -85,B 0,C 180,E1 -4256.743,E2 -4256.743} C_VEL
LIN {X 0,Y 530.983,Z 509.151,A -85,B 0,C 180,E1 -4259.322,E2 -4259.322} C_VEL
LIN {X 0,Y 530.967,Z 509.161,A -85,B 0,C 180,E1 -4262.1,E2 -4262.1} C_VEL
LIN {X 0,Y 530.97,Z 509.152,A -85,B 0,C 180,E1 -4264.85,E2 -4264.85} C_VEL
LIN {X 0,Y 530.965,Z 509.154,A -85,B 0,C 180,E1 -4267.507,E2 -4267.507} C_VEL
LIN {X 0,Y 531.026,Z 509.149,A -85,B 0,C 180,E1 -4270.428,E2 -4270.428} C_VEL
LIN {X 0,Y 530.964,Z 509.154,A -85,B 0,C 180,E1 -4273.493,E2 -4273.493} C_VEL
LIN {X 0,Y 530.962,Z 509.157,A -85,B 0,C 180,E1 -4276.505,E2 -4276.505} C_VEL
LIN {X 0,Y 530.986,Z 509.15,A -85,B 0,C 180,E1 -4278.975,E2 -4278.975} C_VEL
LIN {X 0,Y 530.955,Z 509.155,A -85,B 0,C 180,E1 -4281.529,E2 -4281.529} C_VEL
LIN {X 0,Y 530.978,Z 509.157,A -85,B 0,C 180,E1 -4284.381,E2 -4284.381} C_VEL
LIN {X 0,Y 530.967,Z 509.152,A -85,B 0,C 180,E1 -4287.133,E2 -4287.133} C_VEL
LIN {X 0,Y 530.981,Z 509.154,A -85,B 0,C 180,E1 -4289.803,E2 -4289.803} C_VEL
LIN {X 0,Y 531.012,Z 509.153,A -85,B 0,C 180,E1 -4292.465,E2 -4292.465} C_VEL
LIN {X 0,Y 531.001,Z 509.149,A -85,B 0,C 180,E1 -4294.942,E2 -4294.942} C_VEL
LIN {X 0,Y 530.964,Z 509.161,A -85,B 0,C 180,E1 -4298.246,E2 -4298.246} C_VEL
LIN {X 0,Y 530.99,Z 509.154,A -85,B 0,C 180,E1 -4300.677,E2 -4300.677} C_VEL
LIN {X 0,Y 530.985,Z 509.151,A -85,B 0,C 180,E1 -4303.071,E2 -4303.071} C_VEL
LIN {X 0,Y 531.01,Z 509.147,A -85,B 0,C 180,E1 -4305.435,E2 -4305.435} C_VEL
LIN {X 0,Y 531.04,Z 509.15,A -85,B 0,C 180,E1 -4308.549,E2 -4308.549} C_VEL
LIN {X 0,Y 531.051,Z 509.142,A -85,B 0,C 180,E1 -4311.629,E2 -4311.629} C_VEL
LIN {X 0,Y 531.132,Z 509.137,A -85,B 0,C 180,E1 -4314.685,E2 -4314.685} C_VEL
LIN {X 0,Y 531.131,Z 509.132,A -85,B 0,C 180,E1 -4317.725,E2 -4317.725} C_VEL
LIN {X 0,Y 531.147,Z 509.135,A -85,B 0,C 180,E1 -4320.758,E2 -4320.758} C_VEL
LIN {X 0,Y 531.101,Z 509.138,A -85,B 0,C 180,E1 -4323.034,E2 -4323.034} C_VEL
LIN {X 0,Y 531.075,Z 509.142,A -85,B 0,C 180,E1 -4326.077,E2 -4326.077} C_VEL
LIN {X 0,Y 531.026,Z 509.147,A -85,B 0,C 180,E1 -4329.138,E2 -4329.138} C_VEL
LIN {X 0,Y 531.031,Z 509.148,A -85,B 0,C 180,E1 -4332.225,E2 -4332.225} C_VEL
LIN {X 0,Y 530.987,Z 509.15,A -85,B 0,C 180,E1 -4335.35,E2 -4335.35} C_VEL
LIN {X 0,Y 531.007,Z 509.147,A -85,B 0,C 180,E1 -4337.722,E2 -4337.722} C_VEL
LIN {X 0,Y 530.993,Z 509.154,A -85,B 0,C 180,E1 -4340.938,E2 -4340.938} C_VEL
LIN {X 0,Y 530.971,Z 509.155,A -85,B 0,C 180,E1 -4344.225,E2 -4344.225} C_VEL
LIN {X 0,Y 531.003,Z 509.157,A -85,B 0,C 180,E1 -4346.744,E2 -4346.744} C_VEL
LIN {X 0,Y 530.992,Z 509.151,A -85,B 0,C 180,E1 -4349.322,E2 -4349.322} C_VEL
LIN {X 0,Y 530.972,Z 509.153,A -85,B 0,C 180,E1 -4352.103,E2 -4352.103} C_VEL
LIN {X 0,Y 530.984,Z 509.159,A -85,B 0,C 180,E1 -4354.855,E2 -4354.855} C_VEL
LIN {X 0,Y 530.96,Z 509.154,A -85,B 0,C 180,E1 -4357.508,E2 -4357.508} C_VEL
LIN {X 0,Y 530.978,Z 509.155,A -85,B 0,C 180,E1 -4360.433,E2 -4360.433} C_VEL
LIN {X 0,Y 530.96,Z 509.156,A -85,B 0,C 180,E1 -4363.282,E2 -4363.282} C_VEL
LIN {X 0,Y 530.982,Z 509.151,A -85,B 0,C 180,E1 -4365.621,E2 -4365.621} C_VEL
LIN {X 0,Y 530.996,Z 509.153,A -85,B 0,C 180,E1 -4368.566,E2 -4368.566} C_VEL
LIN {X 0,Y 530.956,Z 509.155,A -85,B 0,C 180,E1 -4371.53,E2 -4371.53} C_VEL
LIN {X 0,Y 530.973,Z 509.155,A -85,B 0,C 180,E1 -4374.382,E2 -4374.382} C_VEL
LIN {X 0,Y 530.969,Z 509.161,A -85,B 0,C 180,E1 -4377.134,E2 -4377.134} C_VEL
LIN {X 0,Y 530.968,Z 509.159,A -85,B 0,C 180,E1 -4379.804,E2 -4379.804} C_VEL
LIN {X 0,Y 530.999,Z 509.222,A -85,B 0,C 180,E1 -4380.746,E2 -4380.746} C_VEL
LIN {X 0,Y 531.688,Z 512.613,A -85,B 0,C 180,E1 -4381.379,E2 -4381.379} C_VEL
LIN {X 0,Y 532.916,Z 519.436,A -85,B 0,C 180,E1 -4382.512,E2 -4382.512} C_VEL
LIN {X 0,Y 532.585,Z 537.092,A -85,B 0,C 180,E1 -4385.189,E2 -4385.189} C_VEL
LIN {X 0,Y 532.226,Z 555.13,A -85,B 0,C 180,E1 -4387.905,E2 -4387.905} C_VEL
LIN {X 0,Y 531.775,Z 573.869,A -85,B 0,C 180,E1 -4390.707,E2 -4390.707} C_VEL
LIN {X 0,Y 531.553,Z 590.532,A -85,B 0,C 180,E1 -4393.09,E2 -4393.09} C_VEL
LIN {X 0,Y 531.247,Z 611.202,A -85,B 0,C 180,E1 -4396.029,E2 -4396.029} C_VEL
LIN {X 0,Y 531.119,Z 626.625,A -85,B 0,C 180,E1 -4398.205,E2 -4398.205} C_VEL
LIN {X 0,Y 531.767,Z 632.407,A -85,B 0,C 180,E1 -4398.328,E2 -4398.328} C_VEL
LIN {X 0,Y 531.755,Z 704.153,A -85,B 0,C 180,E1 -4399.313,E2 -4399.313} C_VEL
LIN {X 0,Y 531.626,Z 713.425,A -85,B 0,C 180,E1 -4399.527,E2 -4399.527} C_VEL
LIN {X 0,Y 531.588,Z 721.897,A -85,B 0,C 180,E1 -4399.815,E2 -4399.815} C_VEL
LIN {X 0,Y 531.417,Z 730.395,A -85,B 0,C 180,E1 -4400.197,E2 -4400.197} C_VEL
LIN {X 0,Y 531.24,Z 738.724,A -85,B 0,C 180,E1 -4400.674,E2 -4400.674} C_VEL
LIN {X 0,Y 531.109,Z 746.766,A -85,B 0,C 180,E1 -4401.247,E2 -4401.247} C_VEL
LIN {X 0,Y 530.929,Z 754.421,A -85,B 0,C 180,E1 -4401.915,E2 -4401.915} C_VEL
LIN {X 0,Y 530.805,Z 762.438,A -85,B 0,C 180,E1 -4402.774,E2 -4402.774} C_VEL
LIN {X 0,Y 530.718,Z 769.421,A -85,B 0,C 180,E1 -4403.725,E2 -4403.725} C_VEL
LIN {X 0,Y 530.543,Z 774.989,A -85,B 0,C 180,E1 -4404.68,E2 -4404.68} C_VEL
LIN {X 0,Y 530.549,Z 780.149,A -85,B 0,C 180,E1 -4405.822,E2 -4405.822} C_VEL
LIN {X 0,Y 530.47,Z 783.937,A -85,B 0,C 180,E1 -4406.962,E2 -4406.962} C_VEL
LIN {X 0,Y 530.411,Z 785.681,A -85,B 0,C 180,E1 -4407.722,E2 -4407.722} C_VEL
LIN {X 0,Y 530.36,Z 786.93,A -85,B 0,C 180,E1 -4408.481,E2 -4408.481} C_VEL
LIN {X 0,Y 530.342,Z 787.707,A -85,B 0,C 180,E1 -4409.241,E2 -4409.241} C_VEL
LIN {X 0,Y 530.34,Z 788,A -85,B 0,C 180,E1 -4410,E2 -4410} C_VEL
LIN {X 0,Y 530.342,Z 787.708,A -85,B 0,C 180,E1 -4410.759,E2 -4410.759} C_VEL
LIN {X 0,Y 530.359,Z 786.931,A -85,B 0,C 180,E1 -4411.519,E2 -4411.519} C_VEL
LIN {X 0,Y 530.411,Z 785.683,A -85,B 0,C 180,E1 -4412.278,E2 -4412.278} C_VEL
LIN {X 0,Y 530.501,Z 782.788,A -85,B 0,C 180,E1 -4413.418,E2 -4413.418} C_VEL
LIN {X 0,Y 530.546,Z 780.149,A -85,B 0,C 180,E1 -4414.178,E2 -4414.178} C_VEL
LIN {X 0,Y 530.543,Z 774.99,A -85,B 0,C 180,E1 -4415.32,E2 -4415.32} C_VEL
LIN {X 0,Y 530.716,Z 769.452,A -85,B 0,C 180,E1 -4416.27,E2 -4416.27} C_VEL
LIN {X 0,Y 530.808,Z 762.439,A -85,B 0,C 180,E1 -4417.226,E2 -4417.226} C_VEL
LIN {X 0,Y 530.929,Z 754.421,A -85,B 0,C 180,E1 -4418.085,E2 -4418.085} C_VEL
LIN {X 0,Y 531.108,Z 746.767,A -85,B 0,C 180,E1 -4418.753,E2 -4418.753} C_VEL
LIN {X 0,Y 531.25,Z 738.727,A -85,B 0,C 180,E1 -4419.326,E2 -4419.326} C_VEL
LIN {X 0,Y 531.429,Z 730.395,A -85,B 0,C 180,E1 -4419.803,E2 -4419.803} C_VEL
LIN {X 0,Y 531.531,Z 721.893,A -85,B 0,C 180,E1 -4420.186,E2 -4420.186} C_VEL
LIN {X 0,Y 531.624,Z 711.76,A -85,B 0,C 180,E1 -4420.521,E2 -4420.521} C_VEL
LIN {X 0,Y 531.81,Z 700.081,A -85,B 0,C 180,E1 -4420.758,E2 -4420.758} C_VEL
LIN {X 0,Y 531.831,Z 632.727,A -85,B 0,C 180,E1 -4421.666,E2 -4421.666} C_VEL
LIN {X 0,Y 531.114,Z 626.801,A -85,B 0,C 180,E1 -4421.779,E2 -4421.779} C_VEL
LIN {X 0,Y 531.124,Z 622.109,A -85,B 0,C 180,E1 -4422.417,E2 -4422.417} C_VEL
LIN {X 0,Y 531.388,Z 601.311,A -85,B 0,C 180,E1 -4425.338,E2 -4425.338} C_VEL
LIN {X 0,Y 531.633,Z 581.306,A -85,B 0,C 180,E1 -4428.124,E2 -4428.124} C_VEL
LIN {X 0,Y 531.941,Z 560.309,A -85,B 0,C 180,E1 -4431.101,E2 -4431.101} C_VEL
LIN {X 0,Y 532.23,Z 540.501,A -85,B 0,C 180,E1 -4433.956,E2 -4433.956} C_VEL
LIN {X 0,Y 532.424,Z 520.773,A -85,B 0,C 180,E1 -4436.878,E2 -4436.878} C_VEL
LIN {X 0,Y 532.403,Z 516.568,A -85,B 0,C 180,E1 -4437.517,E2 -4437.517} C_VEL
LIN {X 0,Y 531.043,Z 509.25,A -85,B 0,C 180,E1 -4438.736,E2 -4438.736} C_VEL
LIN {X 0,Y 530.977,Z 509.154,A -85,B 0,C 180,E1 -4442.102,E2 -4442.102} C_VEL
LIN {X 0,Y 530.979,Z 509.16,A -85,B 0,C 180,E1 -4444.853,E2 -4444.853} C_VEL
LIN {X 0,Y 530.962,Z 509.156,A -85,B 0,C 180,E1 -4447.507,E2 -4447.507} C_VEL
LIN {X 0,Y 530.98,Z 509.154,A -85,B 0,C 180,E1 -4450.432,E2 -4450.432} C_VEL
LIN {X 0,Y 530.966,Z 509.158,A -85,B 0,C 180,E1 -4453.282,E2 -4453.282} C_VEL
LIN {X 0,Y 530.981,Z 509.152,A -85,B 0,C 180,E1 -4455.62,E2 -4455.62} C_VEL
LIN {X 0,Y 531,Z 509.151,A -85,B 0,C 180,E1 -4458.565,E2 -4458.565} C_VEL
LIN {X 0,Y 530.962,Z 509.157,A -85,B 0,C 180,E1 -4461.345,E2 -4461.345} C_VEL
LIN {X 0,Y 530.976,Z 509.153,A -85,B 0,C 180,E1 -4464.382,E2 -4464.382} C_VEL
LIN {X 0,Y 530.967,Z 509.158,A -85,B 0,C 180,E1 -4467.134,E2 -4467.134} C_VEL
LIN {X 0,Y 530.978,Z 509.151,A -85,B 0,C 180,E1 -4469.804,E2 -4469.804} C_VEL
LIN {X 0,Y 531.009,Z 509.151,A -85,B 0,C 180,E1 -4472.466,E2 -4472.466} C_VEL
LIN {X 0,Y 531.003,Z 509.158,A -85,B 0,C 180,E1 -4474.943,E2 -4474.943} C_VEL
LIN {X 0,Y 530.962,Z 509.155,A -85,B 0,C 180,E1 -4478.246,E2 -4478.246} C_VEL
LIN {X 0,Y 530.991,Z 509.155,A -85,B 0,C 180,E1 -4480.677,E2 -4480.677} C_VEL
LIN {X 0,Y 530.984,Z 509.158,A -85,B 0,C 180,E1 -4483.071,E2 -4483.071} C_VEL
LIN {X 0,Y 531.009,Z 509.15,A -85,B 0,C 180,E1 -4485.436,E2 -4485.436} C_VEL
LIN {X 0,Y 531.037,Z 509.15,A -85,B 0,C 180,E1 -4488.55,E2 -4488.55} C_VEL
LIN {X 0,Y 531.052,Z 509.144,A -85,B 0,C 180,E1 -4491.63,E2 -4491.63} C_VEL
LIN {X 0,Y 531.135,Z 509.14,A -85,B 0,C 180,E1 -4494.686,E2 -4494.686} C_VEL
LIN {X 0,Y 531.131,Z 509.134,A -85,B 0,C 180,E1 -4497.725,E2 -4497.725} C_VEL
LIN {X 0,Y 531.148,Z 509.139,A -85,B 0,C 180,E1 -4500.758,E2 -4500.758} C_VEL
LIN {X 0,Y 531.103,Z 509.143,A -85,B 0,C 180,E1 -4503.034,E2 -4503.034} C_VEL
LIN {X 0,Y 531.083,Z 509.144,A -85,B 0,C 180,E1 -4506.077,E2 -4506.077} C_VEL
LIN {X 0,Y 531.093,Z 509.244,A -85,B 0,C 180,E1 -4507.135,E2 -4507.135} C_VEL
LIN {X 0,Y 531.242,Z 510.089,A -85,B 0,C 180,E1 -4507.268,E2 -4507.268} C_VEL
LIN {X 0,Y 532.413,Z 514.136,A -85,B 0,C 180,E1 -4507.371,E2 -4507.371} C_VEL
LIN {X 0,Y 532.337,Z 538.815,A -85,B 0,C 180,E1 -4507.73,E2 -4507.73} C_VEL
LIN {X 0,Y 532.253,Z 552.443,A -85,B 0,C 180,E1 -4508.094,E2 -4508.094} C_VEL
LIN {X 0,Y 532.057,Z 563.935,A -85,B 0,C 180,E1 -4508.546,E2 -4508.546} C_VEL
LIN {X 0,Y 531.914,Z 574.882,A -85,B 0,C 180,E1 -4509.123,E2 -4509.123} C_VEL
LIN {X 0,Y 531.692,Z 585.042,A -85,B 0,C 180,E1 -4509.799,E2 -4509.799} C_VEL
LIN {X 0,Y 531.459,Z 594.512,A -85,B 0,C 180,E1 -4510.573,E2 -4510.573} C_VEL
LIN {X 0,Y 531.247,Z 603.288,A -85,B 0,C 180,E1 -4511.446,E2 -4511.446} C_VEL
LIN {X 0,Y 531.042,Z 612.76,A -85,B 0,C 180,E1 -4512.613,E2 -4512.613} C_VEL
LIN {X 0,Y 530.834,Z 620.271,A -85,B 0,C 180,E1 -4513.787,E2 -4513.787} C_VEL
LIN {X 0,Y 530.742,Z 625.709,A -85,B 0,C 180,E1 -4514.843,E2 -4514.843} C_VEL
LIN {X 0,Y 530.637,Z 629.58,A -85,B 0,C 180,E1 -4515.755,E2 -4515.755} C_VEL
LIN {X 0,Y 530.552,Z 633.525,A -85,B 0,C 180,E1 -4516.944,E2 -4516.944} C_VEL
LIN {X 0,Y 530.511,Z 635.612,A -85,B 0,C 180,E1 -4517.74,E2 -4517.74} C_VEL
LIN {X 0,Y 530.476,Z 637.171,A -85,B 0,C 180,E1 -4518.54,E2 -4518.54} C_VEL
LIN {X 0,Y 530.433,Z 639.001,A -85,B 0,C 180,E1 -4520.151,E2 -4520.151} C_VEL
LIN {X 0,Y 530.433,Z 639.283,A -85,B 0,C 180,E1 -4520.962,E2 -4520.962} C_VEL
LIN {X 0,Y 530.43,Z 638.988,A -85,B 0,C 180,E1 -4521.959,E2 -4521.959} C_VEL
LIN {X 0,Y 530.458,Z 637.377,A -85,B 0,C 180,E1 -4523.42,E2 -4523.42} C_VEL
LIN {X 0,Y 530.545,Z 634.799,A -85,B 0,C 180,E1 -4524.663,E2 -4524.663} C_VEL
LIN {X 0,Y 530.609,Z 631.011,A -85,B 0,C 180,E1 -4525.919,E2 -4525.919} C_VEL
LIN {X 0,Y 530.703,Z 626.189,A -85,B 0,C 180,E1 -4527.118,E2 -4527.118} C_VEL
LIN {X 0,Y 530.84,Z 620.483,A -85,B 0,C 180,E1 -4528.25,E2 -4528.25} C_VEL
LIN {X 0,Y 530.994,Z 613.654,A -85,B 0,C 180,E1 -4529.322,E2 -4529.322} C_VEL
LIN {X 0,Y 531.172,Z 605.785,A -85,B 0,C 180,E1 -4530.343,E2 -4530.343} C_VEL
LIN {X 0,Y 531.409,Z 595.89,A -85,B 0,C 180,E1 -4531.382,E2 -4531.382} C_VEL
LIN {X 0,Y 531.565,Z 588.317,A -85,B 0,C 180,E1 -4532.036,E2 -4532.036} C_VEL
LIN {X 0,Y 531.084,Z 583.56,A -85,B 0,C 180,E1 -4532.411,E2 -4532.411} C_VEL
LIN {X 0,Y 528.494,Z 575.741,A -85,B 0,C 180,E1 -4533.009,E2 -4533.009} C_VEL
LIN {X 0,Y 525.841,Z 567.555,A -85,B 0,C 180,E1 -4533.542,E2 -4533.542} C_VEL
LIN {X 0,Y 525.234,Z 562.226,A -85,B 0,C 180,E1 -4533.81,E2 -4533.81} C_VEL
LIN {X 0,Y 525.41,Z 548.505,A -85,B 0,C 180,E1 -4534.311,E2 -4534.311} C_VEL
LIN {X 0,Y 525.492,Z 535.863,A -85,B 0,C 180,E1 -4534.605,E2 -4534.605} C_VEL
LIN {X 0,Y 525.378,Z 514.868,A -85,B 0,C 180,E1 -4534.908,E2 -4534.908} C_VEL
LIN {X 0,Y 524.096,Z 510.76,A -85,B 0,C 180,E1 -4535.034,E2 -4535.034} C_VEL
LIN {X 0,Y 523.969,Z 510.052,A -85,B 0,C 180,E1 -4535.223,E2 -4535.223} C_VEL
LIN {X 0,Y 523.912,Z 510.035,A -85,B 0,C 180,E1 -4538.103,E2 -4538.103} C_VEL
LIN {X 0,Y 523.958,Z 510.035,A -85,B 0,C 180,E1 -4541.312,E2 -4541.312} C_VEL
LIN {X 0,Y 523.953,Z 510.027,A -85,B 0,C 180,E1 -4544.692,E2 -4544.692} C_VEL
LIN {X 0,Y 523.956,Z 510.028,A -85,B 0,C 180,E1 -4547.883,E2 -4547.883} C_VEL
LIN {X 0,Y 523.977,Z 510.025,A -85,B 0,C 180,E1 -4549.924,E2 -4549.924} C_VEL
LIN {X 0,Y 523.906,Z 510.034,A -85,B 0,C 180,E1 -4552.869,E2 -4552.869} C_VEL
LIN {X 0,Y 523.933,Z 510.034,A -85,B 0,C 180,E1 -4555.711,E2 -4555.711} C_VEL
LIN {X 0,Y 523.924,Z 510.029,A -85,B 0,C 180,E1 -4558.457,E2 -4558.457} C_VEL
LIN {X 0,Y 523.942,Z 510.031,A -85,B 0,C 180,E1 -4561.126,E2 -4561.126} C_VEL
LIN {X 0,Y 523.987,Z 510.025,A -85,B 0,C 180,E1 -4563.981,E2 -4563.981} C_VEL
LIN {X 0,Y 523.928,Z 510.03,A -85,B 0,C 180,E1 -4566.271,E2 -4566.271} C_VEL
LIN {X 0,Y 523.949,Z 510.027,A -85,B 0,C 180,E1 -4568.767,E2 -4568.767} C_VEL
LIN {X 0,Y 523.951,Z 510.03,A -85,B 0,C 180,E1 -4571.221,E2 -4571.221} C_VEL
LIN {X 0,Y 523.934,Z 510.038,A -85,B 0,C 180,E1 -4573.639,E2 -4573.639} C_VEL
LIN {X 0,Y 523.944,Z 510.031,A -85,B 0,C 180,E1 -4576.029,E2 -4576.029} C_VEL
LIN {X 0,Y 524.018,Z 510.018,A -85,B 0,C 180,E1 -4578.395,E2 -4578.395} C_VEL
LIN {X 0,Y 524.006,Z 510.027,A -85,B 0,C 180,E1 -4581.516,E2 -4581.516} C_VEL
LIN {X 0,Y 524.079,Z 510.01,A -85,B 0,C 180,E1 -4584.614,E2 -4584.614} C_VEL
LIN {X 0,Y 524.116,Z 510.015,A -85,B 0,C 180,E1 -4587.695,E2 -4587.695} C_VEL
LIN {X 0,Y 524.126,Z 510.004,A -85,B 0,C 180,E1 -4590.768,E2 -4590.768} C_VEL
LIN {X 0,Y 524.075,Z 510.012,A -85,B 0,C 180,E1 -4593.075,E2 -4593.075} C_VEL
LIN {X 0,Y 524.031,Z 510.02,A -85,B 0,C 180,E1 -4596.159,E2 -4596.159} C_VEL
LIN {X 0,Y 523.998,Z 510.022,A -85,B 0,C 180,E1 -4599.262,E2 -4599.262} C_VEL
LIN {X 0,Y 524.008,Z 510.027,A -85,B 0,C 180,E1 -4601.739,E2 -4601.739} C_VEL
LIN {X 0,Y 523.998,Z 510.021,A -85,B 0,C 180,E1 -4605.052,E2 -4605.052} C_VEL
LIN {X 0,Y 523.968,Z 510.033,A -85,B 0,C 180,E1 -4607.968,E2 -4607.968} C_VEL
LIN {X 0,Y 523.976,Z 510.026,A -85,B 0,C 180,E1 -4610.409,E2 -4610.409} C_VEL
LIN {X 0,Y 523.913,Z 510.031,A -85,B 0,C 180,E1 -4612.893,E2 -4612.893} C_VEL
LIN {X 0,Y 523.987,Z 510.03,A -85,B 0,C 180,E1 -4616.019,E2 -4616.019} C_VEL
LIN {X 0,Y 523.941,Z 510.027,A -85,B 0,C 180,E1 -4618.874,E2 -4618.874} C_VEL
LIN {X 0,Y 523.922,Z 510.033,A -85,B 0,C 180,E1 -4621.543,E2 -4621.543} C_VEL
LIN {X 0,Y 523.933,Z 510.034,A -85,B 0,C 180,E1 -4624.289,E2 -4624.289} C_VEL
LIN {X 0,Y 523.907,Z 510.032,A -85,B 0,C 180,E1 -4627.131,E2 -4627.131} C_VEL
LIN {X 0,Y 523.968,Z 510.033,A -85,B 0,C 180,E1 -4630.133,E2 -4630.133} C_VEL
LIN {X 0,Y 523.923,Z 510.03,A -85,B 0,C 180,E1 -4633.165,E2 -4633.165} C_VEL
LIN {X 0,Y 523.939,Z 510.032,A -85,B 0,C 180,E1 -4635.771,E2 -4635.771} C_VEL
LIN {X 0,Y 523.941,Z 510.028,A -85,B 0,C 180,E1 -4638.907,E2 -4638.907} C_VEL
LIN {X 0,Y 523.913,Z 510.036,A -85,B 0,C 180,E1 -4641.897,E2 -4641.897} C_VEL
LIN {X 0,Y 523.934,Z 510.029,A -85,B 0,C 180,E1 -4644.908,E2 -4644.908} C_VEL
LIN {X 0,Y 523.938,Z 510.03,A -85,B 0,C 180,E1 -4647.677,E2 -4647.677} C_VEL
LIN {X 0,Y 523.964,Z 510.028,A -85,B 0,C 180,E1 -4650.672,E2 -4650.672} C_VEL
LIN {X 0,Y 523.972,Z 510.026,A -85,B 0,C 180,E1 -4653.728,E2 -4653.728} C_VEL
LIN {X 0,Y 523.93,Z 510.039,A -85,B 0,C 180,E1 -4656.27,E2 -4656.27} C_VEL
LIN {X 0,Y 523.94,Z 510.03,A -85,B 0,C 180,E1 -4658.766,E2 -4658.766} C_VEL
LIN {X 0,Y 523.946,Z 510.027,A -85,B 0,C 180,E1 -4661.22,E2 -4661.22} C_VEL
LIN {X 0,Y 523.932,Z 510.029,A -85,B 0,C 180,E1 -4663.638,E2 -4663.638} C_VEL
LIN {X 0,Y 523.932,Z 510.033,A -85,B 0,C 180,E1 -4666.027,E2 -4666.027} C_VEL
LIN {X 0,Y 524.006,Z 510.029,A -85,B 0,C 180,E1 -4668.394,E2 -4668.394} C_VEL
LIN {X 0,Y 523.999,Z 510.02,A -85,B 0,C 180,E1 -4671.516,E2 -4671.516} C_VEL
LIN {X 0,Y 524.09,Z 510.016,A -85,B 0,C 180,E1 -4674.613,E2 -4674.613} C_VEL
LIN {X 0,Y 524.103,Z 510.008,A -85,B 0,C 180,E1 -4677.694,E2 -4677.694} C_VEL
LIN {X 0,Y 524.116,Z 510.011,A -85,B 0,C 180,E1 -4680.768,E2 -4680.768} C_VEL
LIN {X 0,Y 524.067,Z 510.014,A -85,B 0,C 180,E1 -4683.075,E2 -4683.075} C_VEL
LIN {X 0,Y 524.037,Z 510.019,A -85,B 0,C 180,E1 -4686.159,E2 -4686.159} C_VEL
LIN {X 0,Y 523.993,Z 510.022,A -85,B 0,C 180,E1 -4689.262,E2 -4689.262} C_VEL
LIN {X 0,Y 523.993,Z 510.021,A -85,B 0,C 180,E1 -4691.74,E2 -4691.74} C_VEL
LIN {X 0,Y 523.984,Z 510.025,A -85,B 0,C 180,E1 -4695.053,E2 -4695.053} C_VEL
LIN {X 0,Y 523.955,Z 510.027,A -85,B 0,C 180,E1 -4697.969,E2 -4697.969} C_VEL
LIN {X 0,Y 523.963,Z 510.03,A -85,B 0,C 180,E1 -4700.41,E2 -4700.41} C_VEL
LIN {X 0,Y 523.908,Z 510.038,A -85,B 0,C 180,E1 -4702.893,E2 -4702.893} C_VEL
LIN {X 0,Y 523.946,Z 510.027,A -85,B 0,C 180,E1 -4705.419,E2 -4705.419} C_VEL
LIN {X 0,Y 523.963,Z 510.025,A -85,B 0,C 180,E1 -4707.999,E2 -4707.999} C_VEL
LIN {X 0,Y 523.945,Z 510.035,A -85,B 0,C 180,E1 -4710.857,E2 -4710.857} C_VEL
LIN {X 0,Y 523.955,Z 510.026,A -85,B 0,C 180,E1 -4713.736,E2 -4713.736} C_VEL
LIN {X 0,Y 523.916,Z 510.034,A -85,B 0,C 180,E1 -4716.405,E2 -4716.405} C_VEL
LIN {X 0,Y 523.917,Z 510.036,A -85,B 0,C 180,E1 -4719.085,E2 -4719.085} C_VEL
LIN {X 0,Y 523.95,Z 510.027,A -85,B 0,C 180,E1 -4722.119,E2 -4722.119} C_VEL
LIN {X 0,Y 523.95,Z 510.029,A -85,B 0,C 180,E1 -4725.309,E2 -4725.309} C_VEL
LIN {X 0,Y 523.957,Z 510.032,A -85,B 0,C 180,E1 -4728.689,E2 -4728.689} C_VEL
LIN {X 0,Y 523.913,Z 510.031,A -85,B 0,C 180,E1 -4731.899,E2 -4731.899} C_VEL
LIN {X 0,Y 523.931,Z 510.039,A -85,B 0,C 180,E1 -4734.91,E2 -4734.91} C_VEL
LIN {X 0,Y 523.94,Z 510.032,A -85,B 0,C 180,E1 -4737.679,E2 -4737.679} C_VEL
LIN {X 0,Y 523.957,Z 510.14,A -85,B 0,C 180,E1 -4740.561,E2 -4740.561} C_VEL
LIN {X 0,Y 525.922,Z 520.161,A -85,B 0,C 180,E1 -4742.331,E2 -4742.331} C_VEL
LIN {X 0,Y 525.73,Z 532.594,A -85,B 0,C 180,E1 -4744.249,E2 -4744.249} C_VEL
LIN {X 0,Y 525.378,Z 550.297,A -85,B 0,C 180,E1 -4746.966,E2 -4746.966} C_VEL
LIN {X 0,Y 524.833,Z 571.683,A -85,B 0,C 180,E1 -4750.238,E2 -4750.238} C_VEL
LIN {X 0,Y 524.504,Z 591.059,A -85,B 0,C 180,E1 -4753.056,E2 -4753.056} C_VEL
LIN {X 0,Y 524.173,Z 611.727,A -85,B 0,C 180,E1 -4756.035,E2 -4756.035} C_VEL
LIN {X 0,Y 524.064,Z 625.865,A -85,B 0,C 180,E1 -4758.043,E2 -4758.043} C_VEL
LIN {X 0,Y 524.985,Z 636.028,A -85,B 0,C 180,E1 -4758.222,E2 -4758.222} C_VEL
LIN {X 0,Y 524.799,Z 703.781,A -85,B 0,C 180,E1 -4759.17,E2 -4759.17} C_VEL
LIN {X 0,Y 524.61,Z 713.011,A -85,B 0,C 180,E1 -4759.386,E2 -4759.386} C_VEL
LIN {X 0,Y 524.571,Z 722.746,A -85,B 0,C 180,E1 -4759.726,E2 -4759.726} C_VEL
LIN {X 0,Y 524.377,Z 731.977,A -85,B 0,C 180,E1 -4760.161,E2 -4760.161} C_VEL
LIN {X 0,Y 524.183,Z 742.921,A -85,B 0,C 180,E1 -4760.839,E2 -4760.839} C_VEL
LIN {X 0,Y 523.948,Z 751.301,A -85,B 0,C 180,E1 -4761.515,E2 -4761.515} C_VEL
LIN {X 0,Y 523.795,Z 759.032,A -85,B 0,C 180,E1 -4762.289,E2 -4762.289} C_VEL
